REGION Network 79: CmFinalRollerFrontAxisX Position Absolute Position1
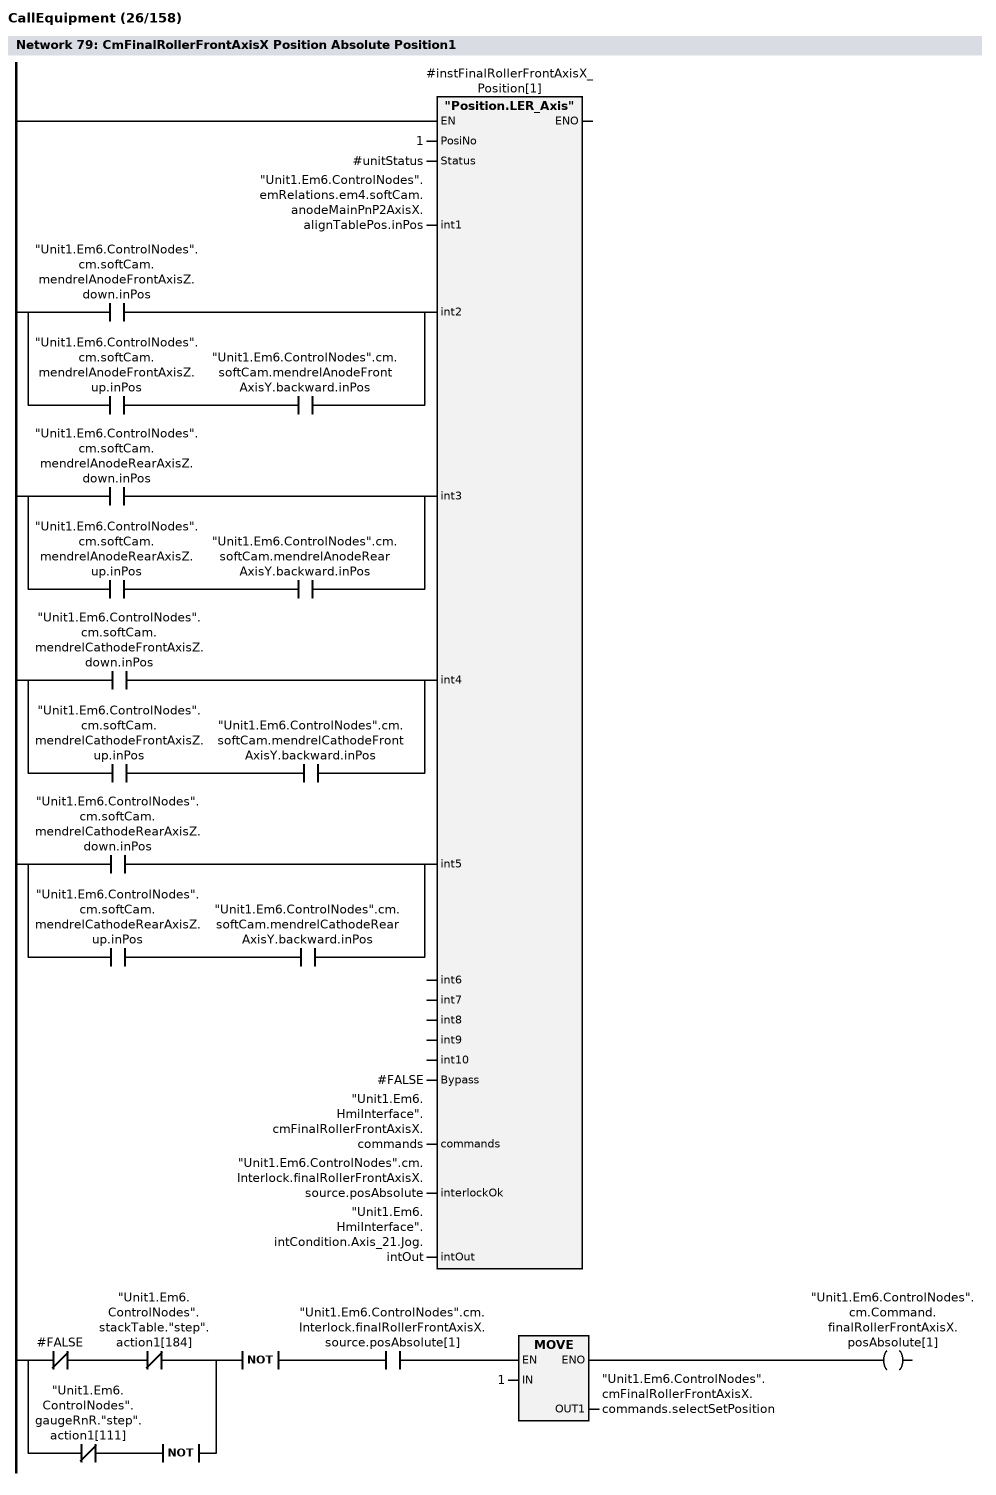
   RUNG wire#powerrail
      #instFinalRollerFrontAxisX_Position[1](int2 := wire#w1, int3 := wire#w2, int4 := wire#w3, int5 := wire#w4, PosiNo := 1, Status := #unitStatus, int1 := "Unit1.Em6.ControlNodes".emRelations.em4.softCam.anodeMainPnP2AxisX.alignTablePos.inPos, int6 :=, int7 :=, int8 :=, int9 :=, int10 :=, Bypass := #FALSE, commands := "Unit1.Em6.HmiInterface".cmFinalRollerFrontAxisX.commands, interlockOk := "Unit1.Em6.ControlNodes".cm.Interlock.finalRollerFrontAxisX.source.posAbsolute, intOut := "Unit1.Em6.HmiInterface".intCondition.Axis_21.Jog.intOut)
   END_RUNG
   RUNG wire#powerrail
      Contact( "Unit1.Em6.ControlNodes".cm.softCam.mendrelAnodeFrontAxisZ.down.inPos )
   END_RUNG wire#w1
   RUNG wire#powerrail
      Contact( "Unit1.Em6.ControlNodes".cm.softCam.mendrelAnodeFrontAxisZ.up.inPos )
      Contact( "Unit1.Em6.ControlNodes".cm.softCam.mendrelAnodeFrontAxisY.backward.inPos )
   END_RUNG wire#w1
   RUNG wire#powerrail
      Contact( "Unit1.Em6.ControlNodes".cm.softCam.mendrelAnodeRearAxisZ.down.inPos )
   END_RUNG wire#w2
   RUNG wire#powerrail
      Contact( "Unit1.Em6.ControlNodes".cm.softCam.mendrelAnodeRearAxisZ.up.inPos )
      Contact( "Unit1.Em6.ControlNodes".cm.softCam.mendrelAnodeRearAxisY.backward.inPos )
   END_RUNG wire#w2
   RUNG wire#powerrail
      Contact( "Unit1.Em6.ControlNodes".cm.softCam.mendrelCathodeFrontAxisZ.down.inPos )
   END_RUNG wire#w3
   RUNG wire#powerrail
      Contact( "Unit1.Em6.ControlNodes".cm.softCam.mendrelCathodeFrontAxisZ.up.inPos )
      Contact( "Unit1.Em6.ControlNodes".cm.softCam.mendrelCathodeFrontAxisY.backward.inPos )
   END_RUNG wire#w3
   RUNG wire#powerrail
      Contact( "Unit1.Em6.ControlNodes".cm.softCam.mendrelCathodeRearAxisZ.down.inPos )
   END_RUNG wire#w4
   RUNG wire#powerrail
      Contact( "Unit1.Em6.ControlNodes".cm.softCam.mendrelCathodeRearAxisZ.up.inPos )
      Contact( "Unit1.Em6.ControlNodes".cm.softCam.mendrelCathodeRearAxisY.backward.inPos )
   END_RUNG wire#w4
   RUNG wire#powerrail
      I_Contact( #FALSE )
      I_Contact( "Unit1.Em6.ControlNodes".stackTable."step".action1[184] )
      wire#w5
      Not()
      Contact( "Unit1.Em6.ControlNodes".cm.Interlock.finalRollerFrontAxisX.source.posAbsolute[1] )
      Move(in := 1, out1 => "Unit1.Em6.ControlNodes".cmFinalRollerFrontAxisX.commands.selectSetPosition)
      Coil( "Unit1.Em6.ControlNodes".cm.Command.finalRollerFrontAxisX.posAbsolute[1] )
   END_RUNG
   RUNG wire#powerrail
      I_Contact( "Unit1.Em6.ControlNodes".gaugeRnR."step".action1[111] )
      Not()
   END_RUNG wire#w5
   // the same network as SCL:
   #instFinalRollerFrontAxisX_Position[1](PosiNo := 1,   // "Position.LER_Axis"
                           Status := #unitStatus,
                           int1 := "Unit1.Em6.ControlNodes".emRelations.em4.softCam.anodeMainPnP2AxisX.alignTablePos.inPos,
                           int2 := "Unit1.Em6.ControlNodes".cm.softCam.mendrelAnodeFrontAxisZ.down.inPos OR ("Unit1.Em6.ControlNodes".cm.softCam.mendrelAnodeFrontAxisZ.up.inPos AND "Unit1.Em6.ControlNodes".cm.softCam.mendrelAnodeFrontAxisY.backward.inPos),
                           int3 := "Unit1.Em6.ControlNodes".cm.softCam.mendrelAnodeRearAxisZ.down.inPos OR ("Unit1.Em6.ControlNodes".cm.softCam.mendrelAnodeRearAxisZ.up.inPos AND "Unit1.Em6.ControlNodes".cm.softCam.mendrelAnodeRearAxisY.backward.inPos),
                           int4 := "Unit1.Em6.ControlNodes".cm.softCam.mendrelCathodeFrontAxisZ.down.inPos OR ("Unit1.Em6.ControlNodes".cm.softCam.mendrelCathodeFrontAxisZ.up.inPos AND "Unit1.Em6.ControlNodes".cm.softCam.mendrelCathodeFrontAxisY.backward.inPos),
                           int5 := "Unit1.Em6.ControlNodes".cm.softCam.mendrelCathodeRearAxisZ.down.inPos OR ("Unit1.Em6.ControlNodes".cm.softCam.mendrelCathodeRearAxisZ.up.inPos AND "Unit1.Em6.ControlNodes".cm.softCam.mendrelCathodeRearAxisY.backward.inPos),
                           Bypass := #FALSE,
                           commands := "Unit1.Em6.HmiInterface".cmFinalRollerFrontAxisX.commands,
                           interlockOk := "Unit1.Em6.ControlNodes".cm.Interlock.finalRollerFrontAxisX.source.posAbsolute,
                           intOut := "Unit1.Em6.HmiInterface".intCondition.Axis_21.Jog.intOut);
   #_w1 := NOT ((NOT #FALSE AND NOT "Unit1.Em6.ControlNodes".stackTable."step".action1[184]) OR NOT (NOT "Unit1.Em6.ControlNodes".gaugeRnR."step".action1[111])) AND "Unit1.Em6.ControlNodes".cm.Interlock.finalRollerFrontAxisX.source.posAbsolute[1];
   IF #_w1 THEN "Unit1.Em6.ControlNodes".cmFinalRollerFrontAxisX.commands.selectSetPosition := 1; END_IF;
   "Unit1.Em6.ControlNodes".cm.Command.finalRollerFrontAxisX.posAbsolute[1] := #_w1;
END_REGION

REGION Network 80: CmFinalRollerFrontAxisX Position Absolute Position2
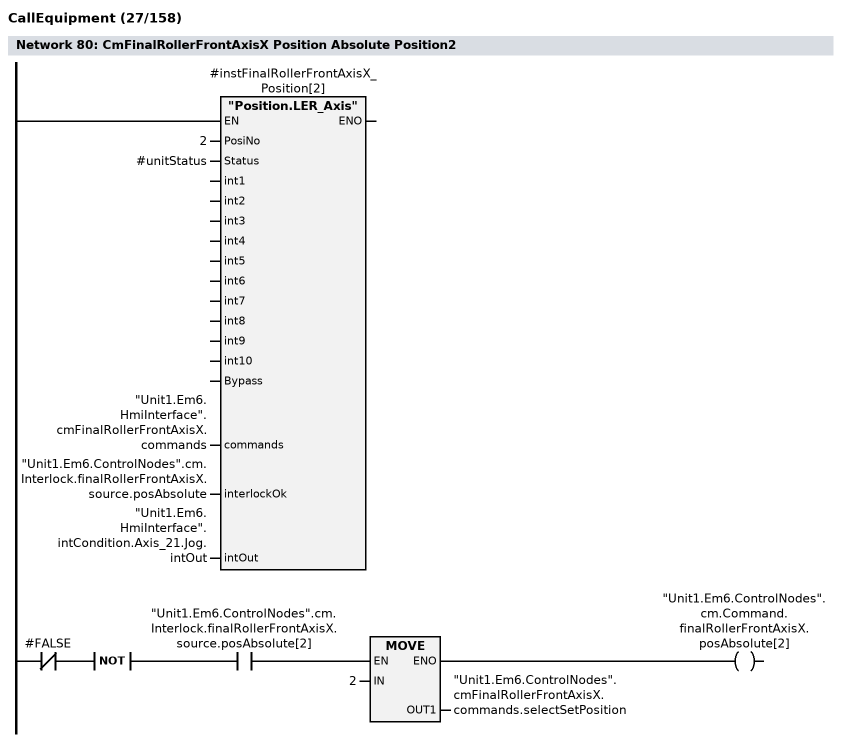
   RUNG wire#powerrail
      #instFinalRollerFrontAxisX_Position[2](PosiNo := 2, Status := #unitStatus, int1 :=, int2 :=, int3 :=, int4 :=, int5 :=, int6 :=, int7 :=, int8 :=, int9 :=, int10 :=, Bypass :=, commands := "Unit1.Em6.HmiInterface".cmFinalRollerFrontAxisX.commands, interlockOk := "Unit1.Em6.ControlNodes".cm.Interlock.finalRollerFrontAxisX.source.posAbsolute, intOut := "Unit1.Em6.HmiInterface".intCondition.Axis_21.Jog.intOut)
   END_RUNG
   RUNG wire#powerrail
      I_Contact( #FALSE )
      Not()
      Contact( "Unit1.Em6.ControlNodes".cm.Interlock.finalRollerFrontAxisX.source.posAbsolute[2] )
      Move(in := 2, out1 => "Unit1.Em6.ControlNodes".cmFinalRollerFrontAxisX.commands.selectSetPosition)
      Coil( "Unit1.Em6.ControlNodes".cm.Command.finalRollerFrontAxisX.posAbsolute[2] )
   END_RUNG
   // the same network as SCL:
   #instFinalRollerFrontAxisX_Position[2](PosiNo := 2,   // "Position.LER_Axis"
                           Status := #unitStatus,
                           commands := "Unit1.Em6.HmiInterface".cmFinalRollerFrontAxisX.commands,
                           interlockOk := "Unit1.Em6.ControlNodes".cm.Interlock.finalRollerFrontAxisX.source.posAbsolute,
                           intOut := "Unit1.Em6.HmiInterface".intCondition.Axis_21.Jog.intOut);
   #_w1 := NOT (NOT #FALSE) AND "Unit1.Em6.ControlNodes".cm.Interlock.finalRollerFrontAxisX.source.posAbsolute[2];
   IF #_w1 THEN "Unit1.Em6.ControlNodes".cmFinalRollerFrontAxisX.commands.selectSetPosition := 2; END_IF;
   "Unit1.Em6.ControlNodes".cm.Command.finalRollerFrontAxisX.posAbsolute[2] := #_w1;
END_REGION

REGION Network 81: CmFinalRollerFrontAxisX Position Absolute Position3
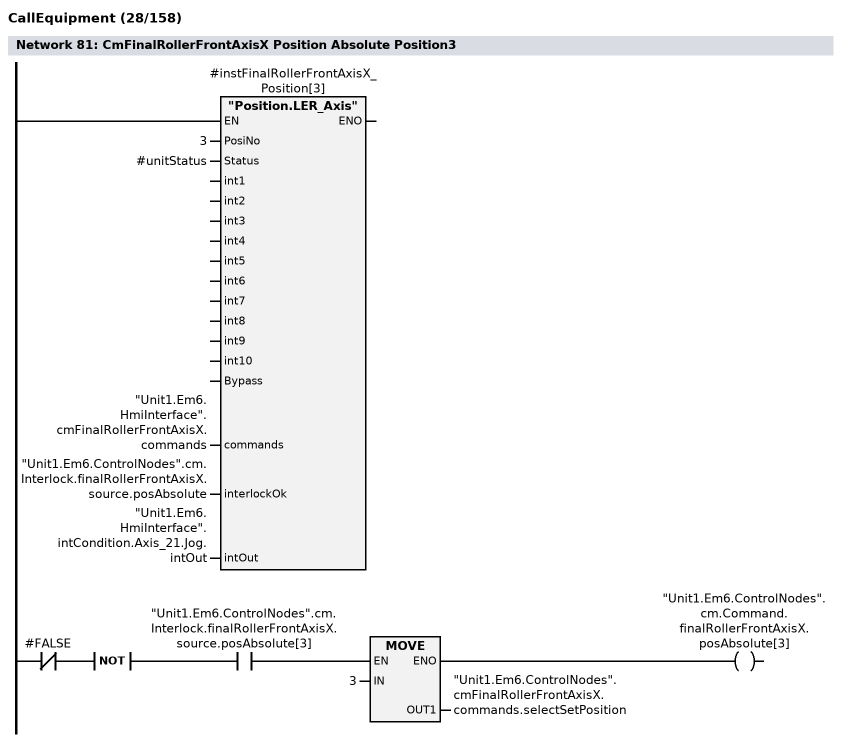
   RUNG wire#powerrail
      #instFinalRollerFrontAxisX_Position[3](PosiNo := 3, Status := #unitStatus, int1 :=, int2 :=, int3 :=, int4 :=, int5 :=, int6 :=, int7 :=, int8 :=, int9 :=, int10 :=, Bypass :=, commands := "Unit1.Em6.HmiInterface".cmFinalRollerFrontAxisX.commands, interlockOk := "Unit1.Em6.ControlNodes".cm.Interlock.finalRollerFrontAxisX.source.posAbsolute, intOut := "Unit1.Em6.HmiInterface".intCondition.Axis_21.Jog.intOut)
   END_RUNG
   RUNG wire#powerrail
      I_Contact( #FALSE )
      Not()
      Contact( "Unit1.Em6.ControlNodes".cm.Interlock.finalRollerFrontAxisX.source.posAbsolute[3] )
      Move(in := 3, out1 => "Unit1.Em6.ControlNodes".cmFinalRollerFrontAxisX.commands.selectSetPosition)
      Coil( "Unit1.Em6.ControlNodes".cm.Command.finalRollerFrontAxisX.posAbsolute[3] )
   END_RUNG
   // the same network as SCL:
   #instFinalRollerFrontAxisX_Position[3](PosiNo := 3,   // "Position.LER_Axis"
                           Status := #unitStatus,
                           commands := "Unit1.Em6.HmiInterface".cmFinalRollerFrontAxisX.commands,
                           interlockOk := "Unit1.Em6.ControlNodes".cm.Interlock.finalRollerFrontAxisX.source.posAbsolute,
                           intOut := "Unit1.Em6.HmiInterface".intCondition.Axis_21.Jog.intOut);
   #_w1 := NOT (NOT #FALSE) AND "Unit1.Em6.ControlNodes".cm.Interlock.finalRollerFrontAxisX.source.posAbsolute[3];
   IF #_w1 THEN "Unit1.Em6.ControlNodes".cmFinalRollerFrontAxisX.commands.selectSetPosition := 3; END_IF;
   "Unit1.Em6.ControlNodes".cm.Command.finalRollerFrontAxisX.posAbsolute[3] := #_w1;
END_REGION

REGION Network 82: CmFinalRollerFrontAxisX Position Absolute Position4
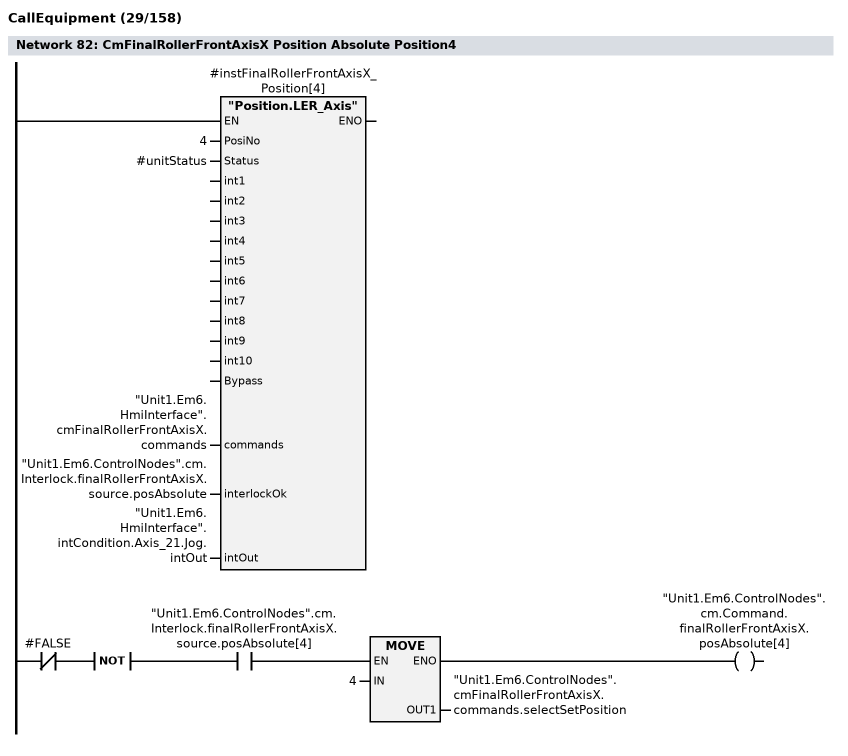
   RUNG wire#powerrail
      #instFinalRollerFrontAxisX_Position[4](PosiNo := 4, Status := #unitStatus, int1 :=, int2 :=, int3 :=, int4 :=, int5 :=, int6 :=, int7 :=, int8 :=, int9 :=, int10 :=, Bypass :=, commands := "Unit1.Em6.HmiInterface".cmFinalRollerFrontAxisX.commands, interlockOk := "Unit1.Em6.ControlNodes".cm.Interlock.finalRollerFrontAxisX.source.posAbsolute, intOut := "Unit1.Em6.HmiInterface".intCondition.Axis_21.Jog.intOut)
   END_RUNG
   RUNG wire#powerrail
      I_Contact( #FALSE )
      Not()
      Contact( "Unit1.Em6.ControlNodes".cm.Interlock.finalRollerFrontAxisX.source.posAbsolute[4] )
      Move(in := 4, out1 => "Unit1.Em6.ControlNodes".cmFinalRollerFrontAxisX.commands.selectSetPosition)
      Coil( "Unit1.Em6.ControlNodes".cm.Command.finalRollerFrontAxisX.posAbsolute[4] )
   END_RUNG
   // the same network as SCL:
   #instFinalRollerFrontAxisX_Position[4](PosiNo := 4,   // "Position.LER_Axis"
                           Status := #unitStatus,
                           commands := "Unit1.Em6.HmiInterface".cmFinalRollerFrontAxisX.commands,
                           interlockOk := "Unit1.Em6.ControlNodes".cm.Interlock.finalRollerFrontAxisX.source.posAbsolute,
                           intOut := "Unit1.Em6.HmiInterface".intCondition.Axis_21.Jog.intOut);
   #_w1 := NOT (NOT #FALSE) AND "Unit1.Em6.ControlNodes".cm.Interlock.finalRollerFrontAxisX.source.posAbsolute[4];
   IF #_w1 THEN "Unit1.Em6.ControlNodes".cmFinalRollerFrontAxisX.commands.selectSetPosition := 4; END_IF;
   "Unit1.Em6.ControlNodes".cm.Command.finalRollerFrontAxisX.posAbsolute[4] := #_w1;
END_REGION

REGION Network 83: CmFinalRollerFrontAxisX Position Absolute Position5
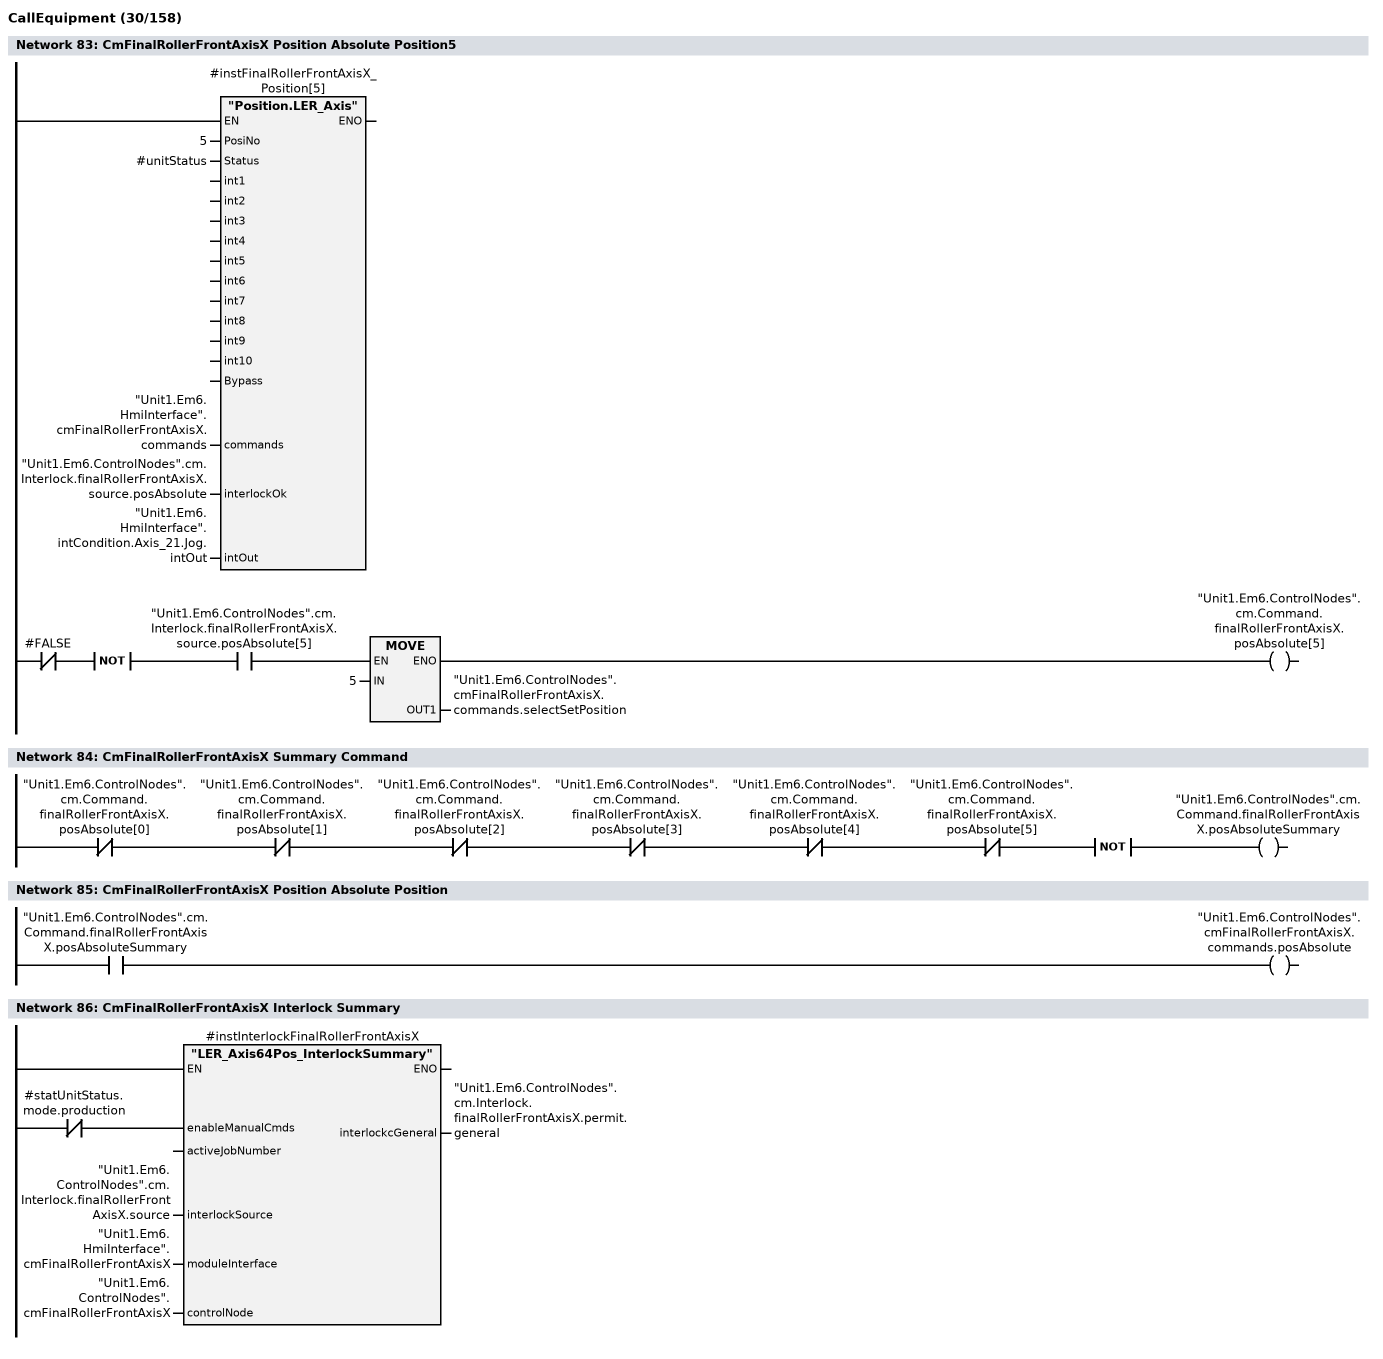
   RUNG wire#powerrail
      #instFinalRollerFrontAxisX_Position[5](PosiNo := 5, Status := #unitStatus, int1 :=, int2 :=, int3 :=, int4 :=, int5 :=, int6 :=, int7 :=, int8 :=, int9 :=, int10 :=, Bypass :=, commands := "Unit1.Em6.HmiInterface".cmFinalRollerFrontAxisX.commands, interlockOk := "Unit1.Em6.ControlNodes".cm.Interlock.finalRollerFrontAxisX.source.posAbsolute, intOut := "Unit1.Em6.HmiInterface".intCondition.Axis_21.Jog.intOut)
   END_RUNG
   RUNG wire#powerrail
      I_Contact( #FALSE )
      Not()
      Contact( "Unit1.Em6.ControlNodes".cm.Interlock.finalRollerFrontAxisX.source.posAbsolute[5] )
      Move(in := 5, out1 => "Unit1.Em6.ControlNodes".cmFinalRollerFrontAxisX.commands.selectSetPosition)
      Coil( "Unit1.Em6.ControlNodes".cm.Command.finalRollerFrontAxisX.posAbsolute[5] )
   END_RUNG
   // the same network as SCL:
   #instFinalRollerFrontAxisX_Position[5](PosiNo := 5,   // "Position.LER_Axis"
                           Status := #unitStatus,
                           commands := "Unit1.Em6.HmiInterface".cmFinalRollerFrontAxisX.commands,
                           interlockOk := "Unit1.Em6.ControlNodes".cm.Interlock.finalRollerFrontAxisX.source.posAbsolute,
                           intOut := "Unit1.Em6.HmiInterface".intCondition.Axis_21.Jog.intOut);
   #_w1 := NOT (NOT #FALSE) AND "Unit1.Em6.ControlNodes".cm.Interlock.finalRollerFrontAxisX.source.posAbsolute[5];
   IF #_w1 THEN "Unit1.Em6.ControlNodes".cmFinalRollerFrontAxisX.commands.selectSetPosition := 5; END_IF;
   "Unit1.Em6.ControlNodes".cm.Command.finalRollerFrontAxisX.posAbsolute[5] := #_w1;
END_REGION

REGION Network 84: CmFinalRollerFrontAxisX Summary Command
   RUNG wire#powerrail
      I_Contact( "Unit1.Em6.ControlNodes".cm.Command.finalRollerFrontAxisX.posAbsolute[0] )
      I_Contact( "Unit1.Em6.ControlNodes".cm.Command.finalRollerFrontAxisX.posAbsolute[1] )
      I_Contact( "Unit1.Em6.ControlNodes".cm.Command.finalRollerFrontAxisX.posAbsolute[2] )
      I_Contact( "Unit1.Em6.ControlNodes".cm.Command.finalRollerFrontAxisX.posAbsolute[3] )
      I_Contact( "Unit1.Em6.ControlNodes".cm.Command.finalRollerFrontAxisX.posAbsolute[4] )
      I_Contact( "Unit1.Em6.ControlNodes".cm.Command.finalRollerFrontAxisX.posAbsolute[5] )
      Not()
      Coil( "Unit1.Em6.ControlNodes".cm.Command.finalRollerFrontAxisX.posAbsoluteSummary )
   END_RUNG
   // the same network as SCL:
   "Unit1.Em6.ControlNodes".cm.Command.finalRollerFrontAxisX.posAbsoluteSummary := NOT (NOT "Unit1.Em6.ControlNodes".cm.Command.finalRollerFrontAxisX.posAbsolute[0] AND NOT "Unit1.Em6.ControlNodes".cm.Command.finalRollerFrontAxisX.posAbsolute[1] AND NOT "Unit1.Em6.ControlNodes".cm.Command.finalRollerFrontAxisX.posAbsolute[2] AND NOT "Unit1.Em6.ControlNodes".cm.Command.finalRollerFrontAxisX.posAbsolute[3] AND NOT "Unit1.Em6.ControlNodes".cm.Command.finalRollerFrontAxisX.posAbsolute[4] AND NOT "Unit1.Em6.ControlNodes".cm.Command.finalRollerFrontAxisX.posAbsolute[5]);
END_REGION

REGION Network 85: CmFinalRollerFrontAxisX Position Absolute Position
   RUNG wire#powerrail
      Contact( "Unit1.Em6.ControlNodes".cm.Command.finalRollerFrontAxisX.posAbsoluteSummary )
      Coil( "Unit1.Em6.ControlNodes".cmFinalRollerFrontAxisX.commands.posAbsolute )
   END_RUNG
   // the same network as SCL:
   "Unit1.Em6.ControlNodes".cmFinalRollerFrontAxisX.commands.posAbsolute := "Unit1.Em6.ControlNodes".cm.Command.finalRollerFrontAxisX.posAbsoluteSummary;
END_REGION

REGION Network 86: CmFinalRollerFrontAxisX Interlock Summary
   RUNG wire#powerrail
      #instInterlockFinalRollerFrontAxisX(enableManualCmds := wire#w1, activeJobNumber :=, interlockSource := "Unit1.Em6.ControlNodes".cm.Interlock.finalRollerFrontAxisX.source, moduleInterface := "Unit1.Em6.HmiInterface".cmFinalRollerFrontAxisX, controlNode := "Unit1.Em6.ControlNodes".cmFinalRollerFrontAxisX, interlockcGeneral => "Unit1.Em6.ControlNodes".cm.Interlock.finalRollerFrontAxisX.permit.general)
   END_RUNG
   RUNG wire#powerrail
      I_Contact( #statUnitStatus.mode.production )
   END_RUNG wire#w1
   // the same network as SCL:
   #instInterlockFinalRollerFrontAxisX(enableManualCmds := NOT #statUnitStatus.mode.production,   // "LER_Axis64Pos_InterlockSummary"
                           interlockSource := "Unit1.Em6.ControlNodes".cm.Interlock.finalRollerFrontAxisX.source,
                           moduleInterface := "Unit1.Em6.HmiInterface".cmFinalRollerFrontAxisX,
                           controlNode := "Unit1.Em6.ControlNodes".cmFinalRollerFrontAxisX,
                           interlockcGeneral => "Unit1.Em6.ControlNodes".cm.Interlock.finalRollerFrontAxisX.permit.general);
END_REGION

REGION Network 87: CmFinalRollerFrontAxisX velocity/speed
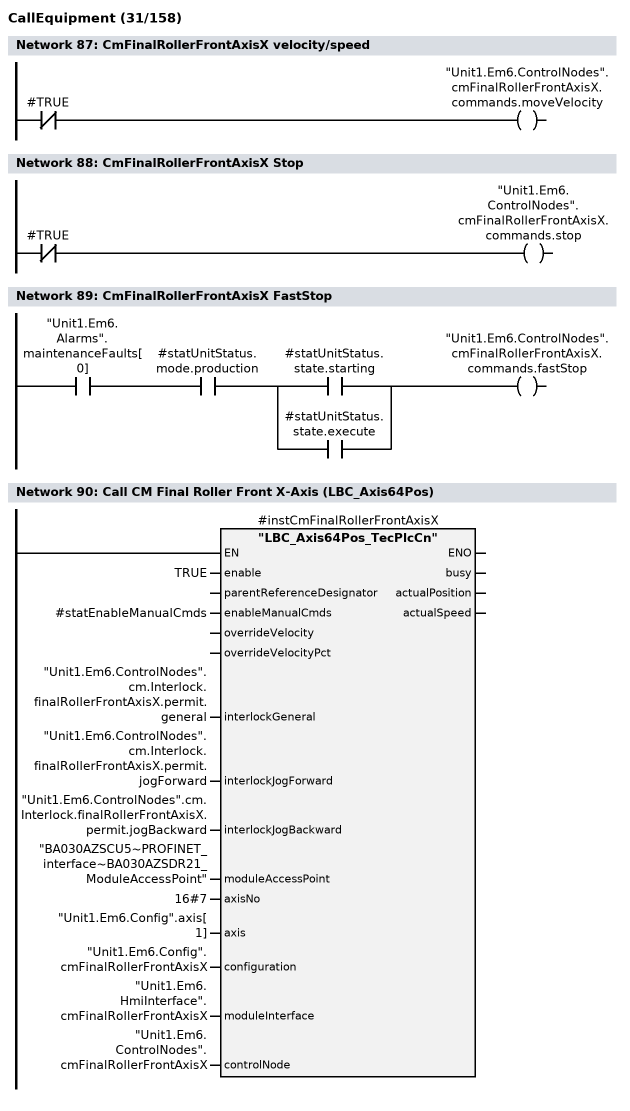
   RUNG wire#powerrail
      I_Contact( #TRUE )
      Coil( "Unit1.Em6.ControlNodes".cmFinalRollerFrontAxisX.commands.moveVelocity )
   END_RUNG
   // the same network as SCL:
   "Unit1.Em6.ControlNodes".cmFinalRollerFrontAxisX.commands.moveVelocity := NOT #TRUE;
END_REGION

REGION Network 88: CmFinalRollerFrontAxisX Stop
   RUNG wire#powerrail
      I_Contact( #TRUE )
      Coil( "Unit1.Em6.ControlNodes".cmFinalRollerFrontAxisX.commands.stop )
   END_RUNG
   // the same network as SCL:
   "Unit1.Em6.ControlNodes".cmFinalRollerFrontAxisX.commands.stop := NOT #TRUE;
END_REGION

REGION Network 89: CmFinalRollerFrontAxisX FastStop
   RUNG wire#powerrail
      Contact( "Unit1.Em6.Alarms".maintenanceFaults[0] )
      Contact( #statUnitStatus.mode.production )
      wire#w1
      Contact( #statUnitStatus.state.starting )
      wire#w2
      Coil( "Unit1.Em6.ControlNodes".cmFinalRollerFrontAxisX.commands.fastStop )
   END_RUNG
   RUNG wire#w1
      Contact( #statUnitStatus.state.execute )
   END_RUNG wire#w2
   // the same network as SCL:
   "Unit1.Em6.ControlNodes".cmFinalRollerFrontAxisX.commands.fastStop := "Unit1.Em6.Alarms".maintenanceFaults[0] AND #statUnitStatus.mode.production AND (#statUnitStatus.state.starting OR #statUnitStatus.state.execute);
END_REGION

REGION Network 90: Call CM Final Roller Front X-Axis (LBC_Axis64Pos)
   RUNG wire#powerrail
      #instCmFinalRollerFrontAxisX(enable := TRUE, parentReferenceDesignator :=, enableManualCmds := #statEnableManualCmds, overrideVelocity :=, overrideVelocityPct :=, interlockGeneral := "Unit1.Em6.ControlNodes".cm.Interlock.finalRollerFrontAxisX.permit.general, interlockJogForward := "Unit1.Em6.ControlNodes".cm.Interlock.finalRollerFrontAxisX.permit.jogForward, interlockJogBackward := "Unit1.Em6.ControlNodes".cm.Interlock.finalRollerFrontAxisX.permit.jogBackward, moduleAccessPoint := "BA030AZSCU5~PROFINET_interface~BA030AZSDR21_ModuleAccessPoint", axisNo := 16#7, axis := "Unit1.Em6.Config".axis[1], configuration := "Unit1.Em6.Config".cmFinalRollerFrontAxisX, moduleInterface := "Unit1.Em6.HmiInterface".cmFinalRollerFrontAxisX, controlNode := "Unit1.Em6.ControlNodes".cmFinalRollerFrontAxisX, busy =>, actualPosition =>, actualSpeed =>)
   END_RUNG
   // the same network as SCL:
   #instCmFinalRollerFrontAxisX(enable := TRUE,   // "LBC_Axis64Pos_TecPlcCn"
                           enableManualCmds := #statEnableManualCmds,
                           interlockGeneral := "Unit1.Em6.ControlNodes".cm.Interlock.finalRollerFrontAxisX.permit.general,
                           interlockJogForward := "Unit1.Em6.ControlNodes".cm.Interlock.finalRollerFrontAxisX.permit.jogForward,
                           interlockJogBackward := "Unit1.Em6.ControlNodes".cm.Interlock.finalRollerFrontAxisX.permit.jogBackward,
                           moduleAccessPoint := "BA030AZSCU5~PROFINET_interface~BA030AZSDR21_ModuleAccessPoint",
                           axisNo := 16#7,
                           axis := "Unit1.Em6.Config".axis[1],
                           configuration := "Unit1.Em6.Config".cmFinalRollerFrontAxisX,
                           moduleInterface := "Unit1.Em6.HmiInterface".cmFinalRollerFrontAxisX,
                           controlNode := "Unit1.Em6.ControlNodes".cmFinalRollerFrontAxisX);
END_REGION

REGION Network 91: CmCathodeMainPnP1AxisX SoftCam
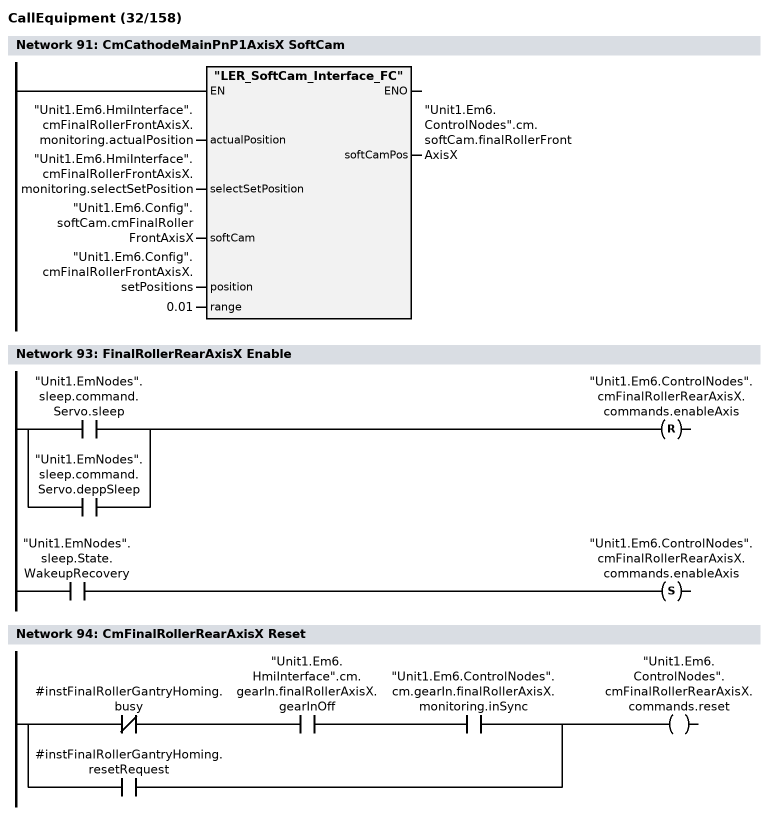
   RUNG wire#powerrail
      "LER_SoftCam_Interface_FC"(actualPosition := "Unit1.Em6.HmiInterface".cmFinalRollerFrontAxisX.monitoring.actualPosition, selectSetPosition := "Unit1.Em6.HmiInterface".cmFinalRollerFrontAxisX.monitoring.selectSetPosition, softCam := "Unit1.Em6.Config".softCam.cmFinalRollerFrontAxisX, position := "Unit1.Em6.Config".cmFinalRollerFrontAxisX.setPositions, range := 0.01, softCamPos => "Unit1.Em6.ControlNodes".cm.softCam.finalRollerFrontAxisX)
   END_RUNG
   // the same network as SCL:
   "LER_SoftCam_Interface_FC"(actualPosition := "Unit1.Em6.HmiInterface".cmFinalRollerFrontAxisX.monitoring.actualPosition,
                           selectSetPosition := "Unit1.Em6.HmiInterface".cmFinalRollerFrontAxisX.monitoring.selectSetPosition,
                           softCam := "Unit1.Em6.Config".softCam.cmFinalRollerFrontAxisX,
                           position := "Unit1.Em6.Config".cmFinalRollerFrontAxisX.setPositions,
                           range := 0.01,
                           softCamPos => "Unit1.Em6.ControlNodes".cm.softCam.finalRollerFrontAxisX);
END_REGION

REGION Network 93: FinalRollerRearAxisX Enable
   RUNG wire#powerrail
      Contact( "Unit1.EmNodes".sleep.command.Servo.sleep )
      wire#w1
      R_Coil( "Unit1.Em6.ControlNodes".cmFinalRollerRearAxisX.commands.enableAxis )
   END_RUNG
   RUNG wire#powerrail
      Contact( "Unit1.EmNodes".sleep.command.Servo.deppSleep )
   END_RUNG wire#w1
   RUNG wire#powerrail
      Contact( "Unit1.EmNodes".sleep.State.WakeupRecovery )
      S_Coil( "Unit1.Em6.ControlNodes".cmFinalRollerRearAxisX.commands.enableAxis )
   END_RUNG
   // the same network as SCL:
   IF "Unit1.EmNodes".sleep.command.Servo.sleep OR "Unit1.EmNodes".sleep.command.Servo.deppSleep THEN
       "Unit1.Em6.ControlNodes".cmFinalRollerRearAxisX.commands.enableAxis := FALSE;
   END_IF;
   IF "Unit1.EmNodes".sleep.State.WakeupRecovery THEN
       "Unit1.Em6.ControlNodes".cmFinalRollerRearAxisX.commands.enableAxis := TRUE;
   END_IF;
END_REGION

REGION Network 94: CmFinalRollerRearAxisX Reset
   RUNG wire#powerrail
      I_Contact( #instFinalRollerGantryHoming.busy )
      Contact( "Unit1.Em6.HmiInterface".cm.gearIn.finalRollerAxisX.gearInOff )
      Contact( "Unit1.Em6.ControlNodes".cm.gearIn.finalRollerAxisX.monitoring.inSync )
      wire#w1
      Coil( "Unit1.Em6.ControlNodes".cmFinalRollerRearAxisX.commands.reset )
   END_RUNG
   RUNG wire#powerrail
      Contact( #instFinalRollerGantryHoming.resetRequest )
   END_RUNG wire#w1
   // the same network as SCL:
   "Unit1.Em6.ControlNodes".cmFinalRollerRearAxisX.commands.reset := (NOT #instFinalRollerGantryHoming.busy AND "Unit1.Em6.HmiInterface".cm.gearIn.finalRollerAxisX.gearInOff AND "Unit1.Em6.ControlNodes".cm.gearIn.finalRollerAxisX.monitoring.inSync) OR #instFinalRollerGantryHoming.resetRequest;
END_REGION

REGION Network 95: CmFinalRollerRearAxisX Home
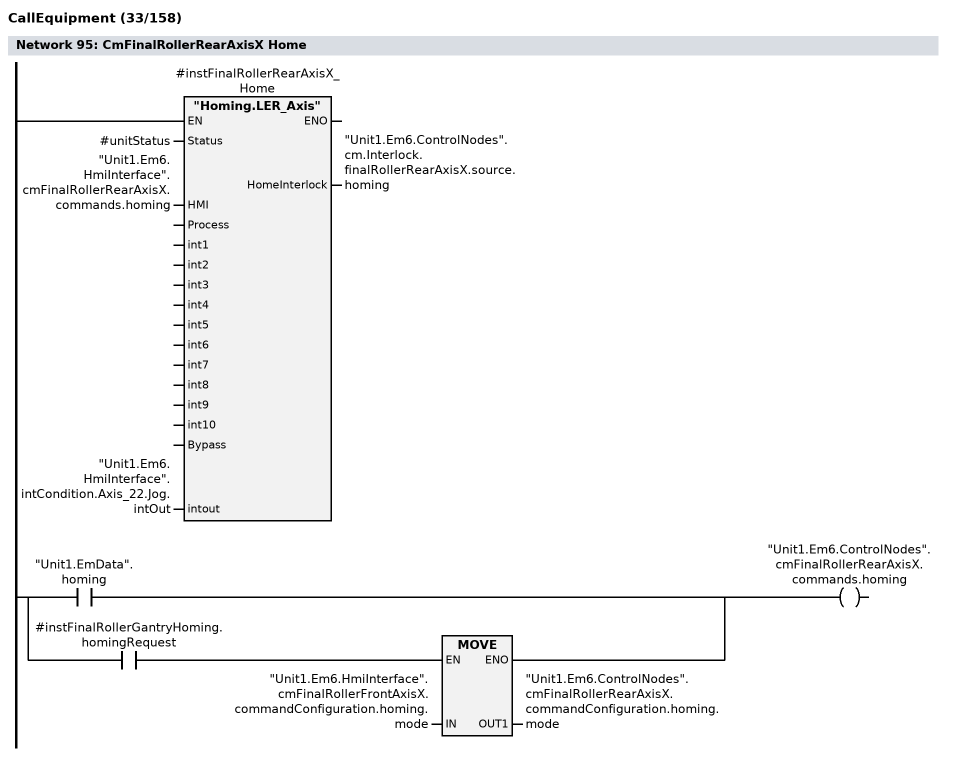
   RUNG wire#powerrail
      #instFinalRollerRearAxisX_Home(Status := #unitStatus, HMI := "Unit1.Em6.HmiInterface".cmFinalRollerRearAxisX.commands.homing, Process :=, int1 :=, int2 :=, int3 :=, int4 :=, int5 :=, int6 :=, int7 :=, int8 :=, int9 :=, int10 :=, Bypass :=, intout := "Unit1.Em6.HmiInterface".intCondition.Axis_22.Jog.intOut, HomeInterlock => "Unit1.Em6.ControlNodes".cm.Interlock.finalRollerRearAxisX.source.homing)
   END_RUNG
   RUNG wire#powerrail
      Contact( "Unit1.EmData".homing )
      wire#w1
      Coil( "Unit1.Em6.ControlNodes".cmFinalRollerRearAxisX.commands.homing )
   END_RUNG
   RUNG wire#powerrail
      Contact( #instFinalRollerGantryHoming.homingRequest )
      Move(in := "Unit1.Em6.HmiInterface".cmFinalRollerFrontAxisX.commandConfiguration.homing.mode, out1 => "Unit1.Em6.ControlNodes".cmFinalRollerRearAxisX.commandConfiguration.homing.mode)
   END_RUNG wire#w1
   // the same network as SCL:
   #instFinalRollerRearAxisX_Home(Status := #unitStatus,   // "Homing.LER_Axis"
                           HMI := "Unit1.Em6.HmiInterface".cmFinalRollerRearAxisX.commands.homing,
                           intout := "Unit1.Em6.HmiInterface".intCondition.Axis_22.Jog.intOut,
                           HomeInterlock => "Unit1.Em6.ControlNodes".cm.Interlock.finalRollerRearAxisX.source.homing);
   IF #instFinalRollerGantryHoming.homingRequest THEN
       "Unit1.Em6.ControlNodes".cmFinalRollerRearAxisX.commandConfiguration.homing.mode := "Unit1.Em6.HmiInterface".cmFinalRollerFrontAxisX.commandConfiguration.homing.mode;
   END_IF;
   "Unit1.Em6.ControlNodes".cmFinalRollerRearAxisX.commands.homing := "Unit1.EmData".homing OR #instFinalRollerGantryHoming.homingRequest;
END_REGION

REGION Network 96: CmFinalRollerRearAxisX Position Absolute Jog
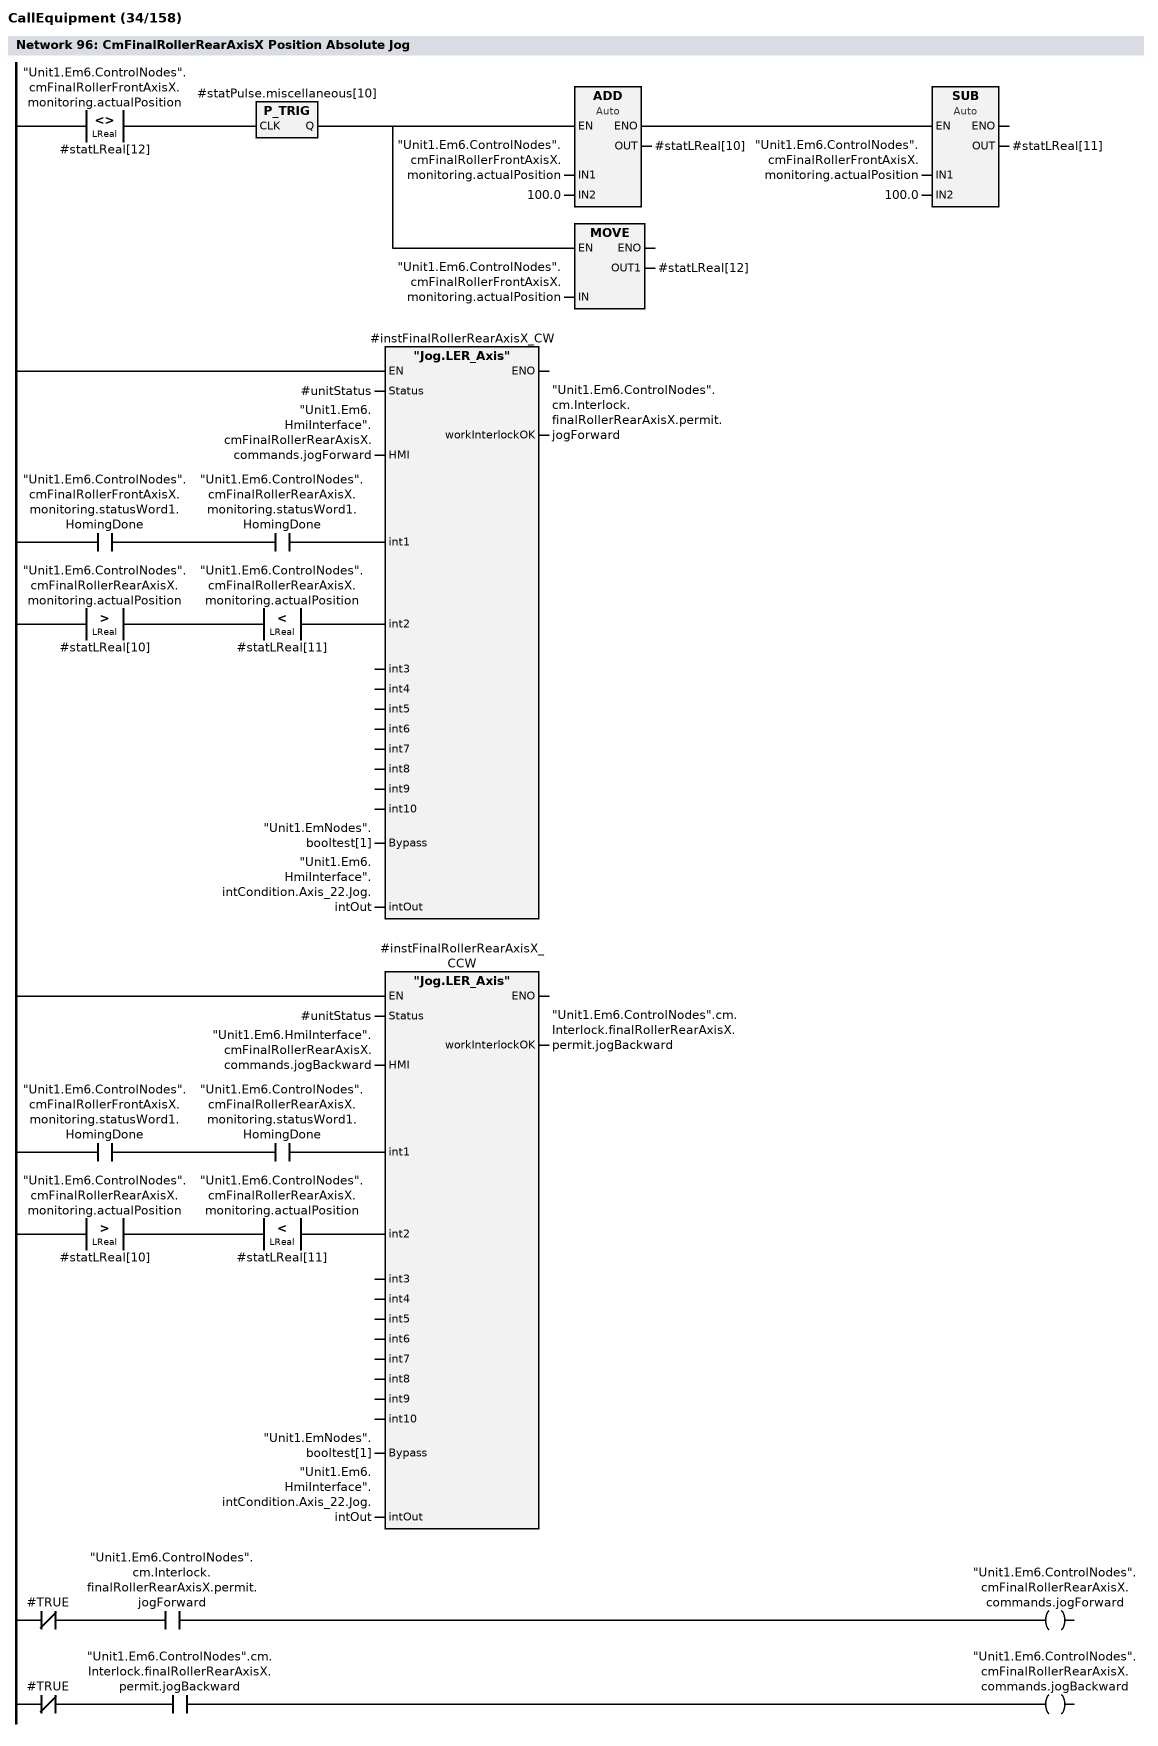
   RUNG wire#powerrail
      { S7_Templates := "SrcType := LReal" } NE_Contact(in1 := "Unit1.Em6.ControlNodes".cmFinalRollerFrontAxisX.monitoring.actualPosition, in2 := #statLReal[12])
      P_Trig( #statPulse.miscellaneous[10] )
      wire#w1
      Add(in1 := "Unit1.Em6.ControlNodes".cmFinalRollerFrontAxisX.monitoring.actualPosition, in2 := 100.0, out => #statLReal[10])
      Sub(in1 := "Unit1.Em6.ControlNodes".cmFinalRollerFrontAxisX.monitoring.actualPosition, in2 := 100.0, out => #statLReal[11])
   END_RUNG
   RUNG wire#w1
      Move(in := "Unit1.Em6.ControlNodes".cmFinalRollerFrontAxisX.monitoring.actualPosition, out1 => #statLReal[12])
   END_RUNG
   RUNG wire#powerrail
      #instFinalRollerRearAxisX_CW(int1 := wire#w2, int2 := wire#w3, Status := #unitStatus, HMI := "Unit1.Em6.HmiInterface".cmFinalRollerRearAxisX.commands.jogForward, int3 :=, int4 :=, int5 :=, int6 :=, int7 :=, int8 :=, int9 :=, int10 :=, Bypass := "Unit1.EmNodes".booltest[1], intOut := "Unit1.Em6.HmiInterface".intCondition.Axis_22.Jog.intOut, workInterlockOK => "Unit1.Em6.ControlNodes".cm.Interlock.finalRollerRearAxisX.permit.jogForward)
   END_RUNG
   RUNG wire#powerrail
      Contact( "Unit1.Em6.ControlNodes".cmFinalRollerFrontAxisX.monitoring.statusWord1.HomingDone )
      Contact( "Unit1.Em6.ControlNodes".cmFinalRollerRearAxisX.monitoring.statusWord1.HomingDone )
   END_RUNG wire#w2
   RUNG wire#powerrail
      { S7_Templates := "SrcType := LReal" } GT_Contact(in1 := "Unit1.Em6.ControlNodes".cmFinalRollerRearAxisX.monitoring.actualPosition, in2 := #statLReal[10])
      { S7_Templates := "SrcType := LReal" } LT_Contact(in1 := "Unit1.Em6.ControlNodes".cmFinalRollerRearAxisX.monitoring.actualPosition, in2 := #statLReal[11])
   END_RUNG wire#w3
   RUNG wire#powerrail
      #instFinalRollerRearAxisX_CCW(int1 := wire#w4, int2 := wire#w5, Status := #unitStatus, HMI := "Unit1.Em6.HmiInterface".cmFinalRollerRearAxisX.commands.jogBackward, int3 :=, int4 :=, int5 :=, int6 :=, int7 :=, int8 :=, int9 :=, int10 :=, Bypass := "Unit1.EmNodes".booltest[1], intOut := "Unit1.Em6.HmiInterface".intCondition.Axis_22.Jog.intOut, workInterlockOK => "Unit1.Em6.ControlNodes".cm.Interlock.finalRollerRearAxisX.permit.jogBackward)
   END_RUNG
   RUNG wire#powerrail
      Contact( "Unit1.Em6.ControlNodes".cmFinalRollerFrontAxisX.monitoring.statusWord1.HomingDone )
      Contact( "Unit1.Em6.ControlNodes".cmFinalRollerRearAxisX.monitoring.statusWord1.HomingDone )
   END_RUNG wire#w4
   RUNG wire#powerrail
      { S7_Templates := "SrcType := LReal" } GT_Contact(in1 := "Unit1.Em6.ControlNodes".cmFinalRollerRearAxisX.monitoring.actualPosition, in2 := #statLReal[10])
      { S7_Templates := "SrcType := LReal" } LT_Contact(in1 := "Unit1.Em6.ControlNodes".cmFinalRollerRearAxisX.monitoring.actualPosition, in2 := #statLReal[11])
   END_RUNG wire#w5
   RUNG wire#powerrail
      I_Contact( #TRUE )
      Contact( "Unit1.Em6.ControlNodes".cm.Interlock.finalRollerRearAxisX.permit.jogForward )
      Coil( "Unit1.Em6.ControlNodes".cmFinalRollerRearAxisX.commands.jogForward )
   END_RUNG
   RUNG wire#powerrail
      I_Contact( #TRUE )
      Contact( "Unit1.Em6.ControlNodes".cm.Interlock.finalRollerRearAxisX.permit.jogBackward )
      Coil( "Unit1.Em6.ControlNodes".cmFinalRollerRearAxisX.commands.jogBackward )
   END_RUNG
   // the same network as SCL:
   #_w1 := "Unit1.Em6.ControlNodes".cmFinalRollerFrontAxisX.monitoring.actualPosition <> #statLReal[12];
   #_w2 := #_w1 AND NOT #statPulse.miscellaneous[10];   // rising edge
   #statPulse.miscellaneous[10] := #_w1;
   IF #_w2 THEN
       #statLReal[10] := "Unit1.Em6.ControlNodes".cmFinalRollerFrontAxisX.monitoring.actualPosition + 100.0;
       #statLReal[11] := "Unit1.Em6.ControlNodes".cmFinalRollerFrontAxisX.monitoring.actualPosition - 100.0;
       #statLReal[12] := "Unit1.Em6.ControlNodes".cmFinalRollerFrontAxisX.monitoring.actualPosition;
   END_IF;
   #instFinalRollerRearAxisX_CW(Status := #unitStatus,   // "Jog.LER_Axis"
                           HMI := "Unit1.Em6.HmiInterface".cmFinalRollerRearAxisX.commands.jogForward,
                           int1 := "Unit1.Em6.ControlNodes".cmFinalRollerFrontAxisX.monitoring.statusWord1.HomingDone AND "Unit1.Em6.ControlNodes".cmFinalRollerRearAxisX.monitoring.statusWord1.HomingDone,
                           int2 := ("Unit1.Em6.ControlNodes".cmFinalRollerRearAxisX.monitoring.actualPosition > #statLReal[10]) AND ("Unit1.Em6.ControlNodes".cmFinalRollerRearAxisX.monitoring.actualPosition < #statLReal[11]),
                           Bypass := "Unit1.EmNodes".booltest[1],
                           intOut := "Unit1.Em6.HmiInterface".intCondition.Axis_22.Jog.intOut,
                           workInterlockOK => "Unit1.Em6.ControlNodes".cm.Interlock.finalRollerRearAxisX.permit.jogForward);
   #instFinalRollerRearAxisX_CCW(Status := #unitStatus,   // "Jog.LER_Axis"
                           HMI := "Unit1.Em6.HmiInterface".cmFinalRollerRearAxisX.commands.jogBackward,
                           int1 := "Unit1.Em6.ControlNodes".cmFinalRollerFrontAxisX.monitoring.statusWord1.HomingDone AND "Unit1.Em6.ControlNodes".cmFinalRollerRearAxisX.monitoring.statusWord1.HomingDone,
                           int2 := ("Unit1.Em6.ControlNodes".cmFinalRollerRearAxisX.monitoring.actualPosition > #statLReal[10]) AND ("Unit1.Em6.ControlNodes".cmFinalRollerRearAxisX.monitoring.actualPosition < #statLReal[11]),
                           Bypass := "Unit1.EmNodes".booltest[1],
                           intOut := "Unit1.Em6.HmiInterface".intCondition.Axis_22.Jog.intOut,
                           workInterlockOK => "Unit1.Em6.ControlNodes".cm.Interlock.finalRollerRearAxisX.permit.jogBackward);
   "Unit1.Em6.ControlNodes".cmFinalRollerRearAxisX.commands.jogForward := NOT #TRUE AND "Unit1.Em6.ControlNodes".cm.Interlock.finalRollerRearAxisX.permit.jogForward;
   "Unit1.Em6.ControlNodes".cmFinalRollerRearAxisX.commands.jogBackward := NOT #TRUE AND "Unit1.Em6.ControlNodes".cm.Interlock.finalRollerRearAxisX.permit.jogBackward;
END_REGION

REGION Network 97: CmFinalRollerRearAxisX Position Absolute Position0
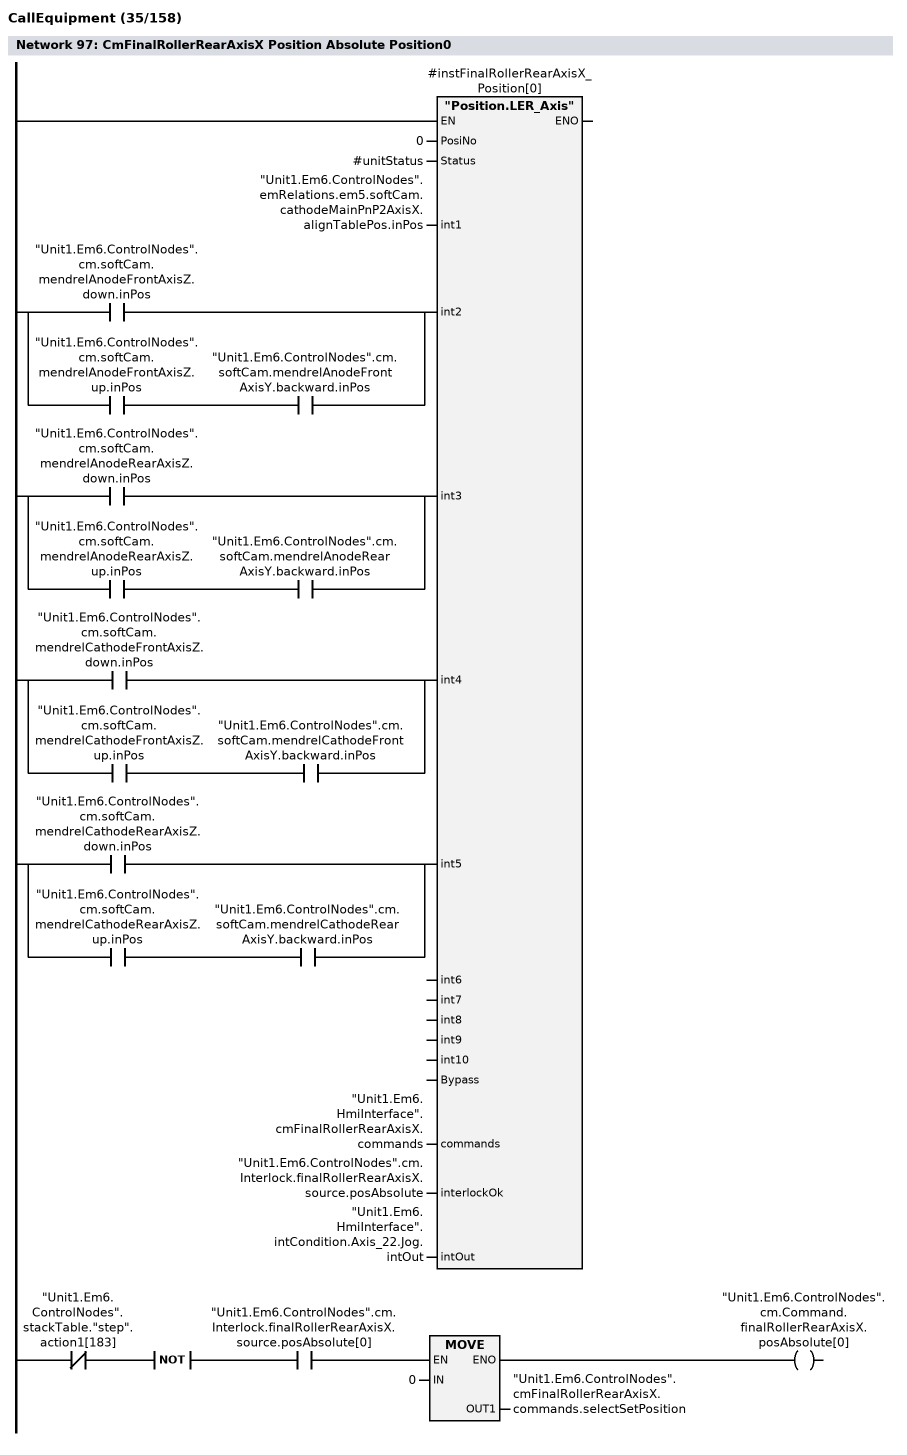
   RUNG wire#powerrail
      #instFinalRollerRearAxisX_Position[0](int2 := wire#w1, int3 := wire#w2, int4 := wire#w3, int5 := wire#w4, PosiNo := 0, Status := #unitStatus, int1 := "Unit1.Em6.ControlNodes".emRelations.em5.softCam.cathodeMainPnP2AxisX.alignTablePos.inPos, int6 :=, int7 :=, int8 :=, int9 :=, int10 :=, Bypass :=, commands := "Unit1.Em6.HmiInterface".cmFinalRollerRearAxisX.commands, interlockOk := "Unit1.Em6.ControlNodes".cm.Interlock.finalRollerRearAxisX.source.posAbsolute, intOut := "Unit1.Em6.HmiInterface".intCondition.Axis_22.Jog.intOut)
   END_RUNG
   RUNG wire#powerrail
      Contact( "Unit1.Em6.ControlNodes".cm.softCam.mendrelAnodeFrontAxisZ.down.inPos )
   END_RUNG wire#w1
   RUNG wire#powerrail
      Contact( "Unit1.Em6.ControlNodes".cm.softCam.mendrelAnodeFrontAxisZ.up.inPos )
      Contact( "Unit1.Em6.ControlNodes".cm.softCam.mendrelAnodeFrontAxisY.backward.inPos )
   END_RUNG wire#w1
   RUNG wire#powerrail
      Contact( "Unit1.Em6.ControlNodes".cm.softCam.mendrelAnodeRearAxisZ.down.inPos )
   END_RUNG wire#w2
   RUNG wire#powerrail
      Contact( "Unit1.Em6.ControlNodes".cm.softCam.mendrelAnodeRearAxisZ.up.inPos )
      Contact( "Unit1.Em6.ControlNodes".cm.softCam.mendrelAnodeRearAxisY.backward.inPos )
   END_RUNG wire#w2
   RUNG wire#powerrail
      Contact( "Unit1.Em6.ControlNodes".cm.softCam.mendrelCathodeFrontAxisZ.down.inPos )
   END_RUNG wire#w3
   RUNG wire#powerrail
      Contact( "Unit1.Em6.ControlNodes".cm.softCam.mendrelCathodeFrontAxisZ.up.inPos )
      Contact( "Unit1.Em6.ControlNodes".cm.softCam.mendrelCathodeFrontAxisY.backward.inPos )
   END_RUNG wire#w3
   RUNG wire#powerrail
      Contact( "Unit1.Em6.ControlNodes".cm.softCam.mendrelCathodeRearAxisZ.down.inPos )
   END_RUNG wire#w4
   RUNG wire#powerrail
      Contact( "Unit1.Em6.ControlNodes".cm.softCam.mendrelCathodeRearAxisZ.up.inPos )
      Contact( "Unit1.Em6.ControlNodes".cm.softCam.mendrelCathodeRearAxisY.backward.inPos )
   END_RUNG wire#w4
   RUNG wire#powerrail
      I_Contact( "Unit1.Em6.ControlNodes".stackTable."step".action1[183] )
      Not()
      Contact( "Unit1.Em6.ControlNodes".cm.Interlock.finalRollerRearAxisX.source.posAbsolute[0] )
      Move(in := 0, out1 => "Unit1.Em6.ControlNodes".cmFinalRollerRearAxisX.commands.selectSetPosition)
      Coil( "Unit1.Em6.ControlNodes".cm.Command.finalRollerRearAxisX.posAbsolute[0] )
   END_RUNG
   // the same network as SCL:
   #instFinalRollerRearAxisX_Position[0](PosiNo := 0,   // "Position.LER_Axis"
                           Status := #unitStatus,
                           int1 := "Unit1.Em6.ControlNodes".emRelations.em5.softCam.cathodeMainPnP2AxisX.alignTablePos.inPos,
                           int2 := "Unit1.Em6.ControlNodes".cm.softCam.mendrelAnodeFrontAxisZ.down.inPos OR ("Unit1.Em6.ControlNodes".cm.softCam.mendrelAnodeFrontAxisZ.up.inPos AND "Unit1.Em6.ControlNodes".cm.softCam.mendrelAnodeFrontAxisY.backward.inPos),
                           int3 := "Unit1.Em6.ControlNodes".cm.softCam.mendrelAnodeRearAxisZ.down.inPos OR ("Unit1.Em6.ControlNodes".cm.softCam.mendrelAnodeRearAxisZ.up.inPos AND "Unit1.Em6.ControlNodes".cm.softCam.mendrelAnodeRearAxisY.backward.inPos),
                           int4 := "Unit1.Em6.ControlNodes".cm.softCam.mendrelCathodeFrontAxisZ.down.inPos OR ("Unit1.Em6.ControlNodes".cm.softCam.mendrelCathodeFrontAxisZ.up.inPos AND "Unit1.Em6.ControlNodes".cm.softCam.mendrelCathodeFrontAxisY.backward.inPos),
                           int5 := "Unit1.Em6.ControlNodes".cm.softCam.mendrelCathodeRearAxisZ.down.inPos OR ("Unit1.Em6.ControlNodes".cm.softCam.mendrelCathodeRearAxisZ.up.inPos AND "Unit1.Em6.ControlNodes".cm.softCam.mendrelCathodeRearAxisY.backward.inPos),
                           commands := "Unit1.Em6.HmiInterface".cmFinalRollerRearAxisX.commands,
                           interlockOk := "Unit1.Em6.ControlNodes".cm.Interlock.finalRollerRearAxisX.source.posAbsolute,
                           intOut := "Unit1.Em6.HmiInterface".intCondition.Axis_22.Jog.intOut);
   #_w1 := NOT (NOT "Unit1.Em6.ControlNodes".stackTable."step".action1[183]) AND "Unit1.Em6.ControlNodes".cm.Interlock.finalRollerRearAxisX.source.posAbsolute[0];
   IF #_w1 THEN "Unit1.Em6.ControlNodes".cmFinalRollerRearAxisX.commands.selectSetPosition := 0; END_IF;
   "Unit1.Em6.ControlNodes".cm.Command.finalRollerRearAxisX.posAbsolute[0] := #_w1;
END_REGION

REGION Network 98: CmFinalRollerRearAxisX Position Absolute Position1
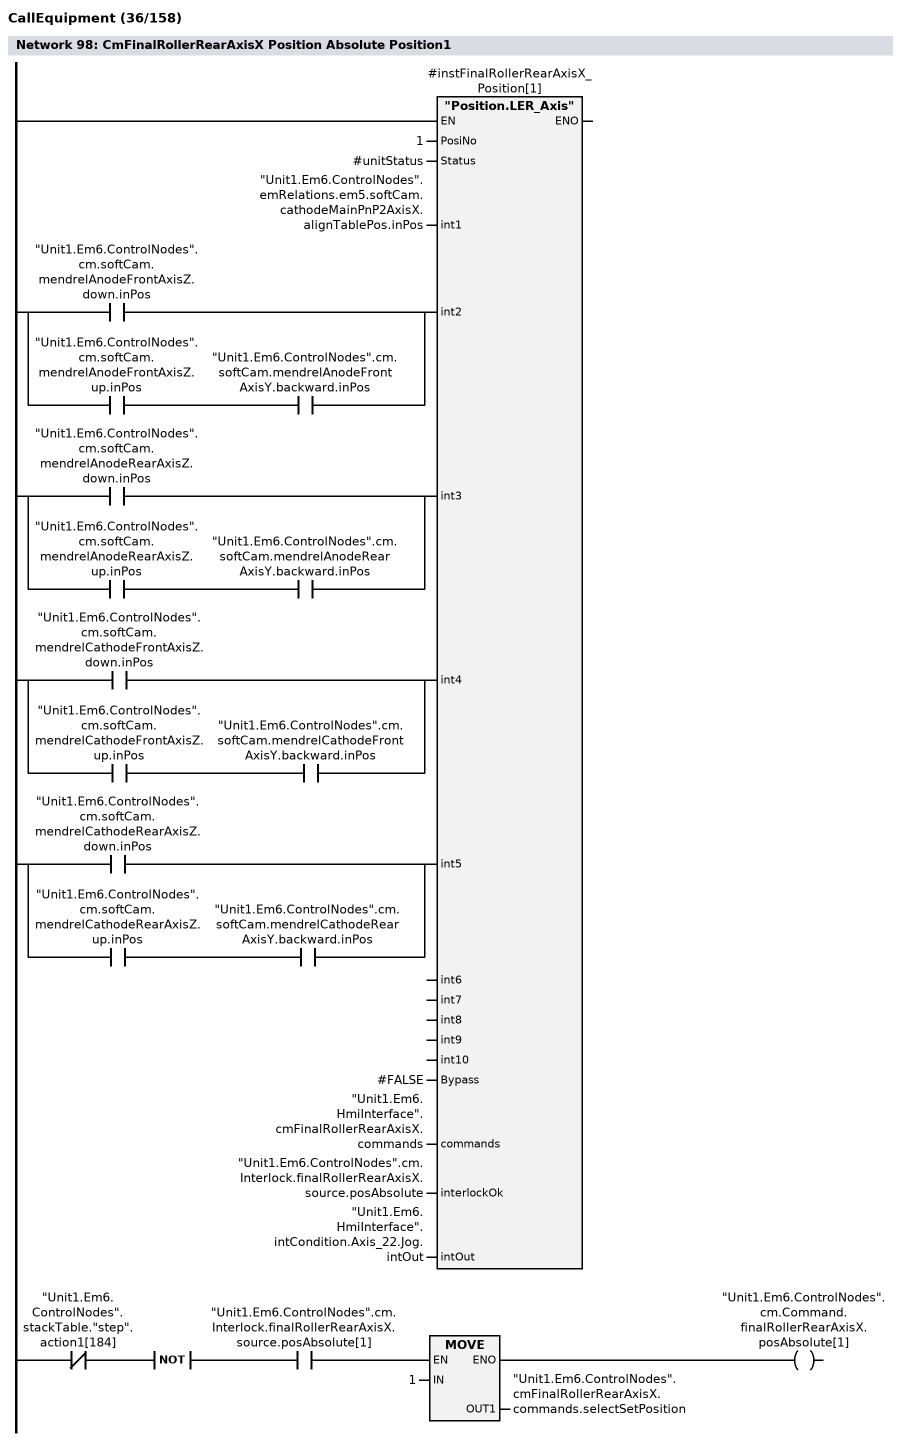
   RUNG wire#powerrail
      #instFinalRollerRearAxisX_Position[1](int2 := wire#w1, int3 := wire#w2, int4 := wire#w3, int5 := wire#w4, PosiNo := 1, Status := #unitStatus, int1 := "Unit1.Em6.ControlNodes".emRelations.em5.softCam.cathodeMainPnP2AxisX.alignTablePos.inPos, int6 :=, int7 :=, int8 :=, int9 :=, int10 :=, Bypass := #FALSE, commands := "Unit1.Em6.HmiInterface".cmFinalRollerRearAxisX.commands, interlockOk := "Unit1.Em6.ControlNodes".cm.Interlock.finalRollerRearAxisX.source.posAbsolute, intOut := "Unit1.Em6.HmiInterface".intCondition.Axis_22.Jog.intOut)
   END_RUNG
   RUNG wire#powerrail
      Contact( "Unit1.Em6.ControlNodes".cm.softCam.mendrelAnodeFrontAxisZ.down.inPos )
   END_RUNG wire#w1
   RUNG wire#powerrail
      Contact( "Unit1.Em6.ControlNodes".cm.softCam.mendrelAnodeFrontAxisZ.up.inPos )
      Contact( "Unit1.Em6.ControlNodes".cm.softCam.mendrelAnodeFrontAxisY.backward.inPos )
   END_RUNG wire#w1
   RUNG wire#powerrail
      Contact( "Unit1.Em6.ControlNodes".cm.softCam.mendrelAnodeRearAxisZ.down.inPos )
   END_RUNG wire#w2
   RUNG wire#powerrail
      Contact( "Unit1.Em6.ControlNodes".cm.softCam.mendrelAnodeRearAxisZ.up.inPos )
      Contact( "Unit1.Em6.ControlNodes".cm.softCam.mendrelAnodeRearAxisY.backward.inPos )
   END_RUNG wire#w2
   RUNG wire#powerrail
      Contact( "Unit1.Em6.ControlNodes".cm.softCam.mendrelCathodeFrontAxisZ.down.inPos )
   END_RUNG wire#w3
   RUNG wire#powerrail
      Contact( "Unit1.Em6.ControlNodes".cm.softCam.mendrelCathodeFrontAxisZ.up.inPos )
      Contact( "Unit1.Em6.ControlNodes".cm.softCam.mendrelCathodeFrontAxisY.backward.inPos )
   END_RUNG wire#w3
   RUNG wire#powerrail
      Contact( "Unit1.Em6.ControlNodes".cm.softCam.mendrelCathodeRearAxisZ.down.inPos )
   END_RUNG wire#w4
   RUNG wire#powerrail
      Contact( "Unit1.Em6.ControlNodes".cm.softCam.mendrelCathodeRearAxisZ.up.inPos )
      Contact( "Unit1.Em6.ControlNodes".cm.softCam.mendrelCathodeRearAxisY.backward.inPos )
   END_RUNG wire#w4
   RUNG wire#powerrail
      I_Contact( "Unit1.Em6.ControlNodes".stackTable."step".action1[184] )
      Not()
      Contact( "Unit1.Em6.ControlNodes".cm.Interlock.finalRollerRearAxisX.source.posAbsolute[1] )
      Move(in := 1, out1 => "Unit1.Em6.ControlNodes".cmFinalRollerRearAxisX.commands.selectSetPosition)
      Coil( "Unit1.Em6.ControlNodes".cm.Command.finalRollerRearAxisX.posAbsolute[1] )
   END_RUNG
   // the same network as SCL:
   #instFinalRollerRearAxisX_Position[1](PosiNo := 1,   // "Position.LER_Axis"
                           Status := #unitStatus,
                           int1 := "Unit1.Em6.ControlNodes".emRelations.em5.softCam.cathodeMainPnP2AxisX.alignTablePos.inPos,
                           int2 := "Unit1.Em6.ControlNodes".cm.softCam.mendrelAnodeFrontAxisZ.down.inPos OR ("Unit1.Em6.ControlNodes".cm.softCam.mendrelAnodeFrontAxisZ.up.inPos AND "Unit1.Em6.ControlNodes".cm.softCam.mendrelAnodeFrontAxisY.backward.inPos),
                           int3 := "Unit1.Em6.ControlNodes".cm.softCam.mendrelAnodeRearAxisZ.down.inPos OR ("Unit1.Em6.ControlNodes".cm.softCam.mendrelAnodeRearAxisZ.up.inPos AND "Unit1.Em6.ControlNodes".cm.softCam.mendrelAnodeRearAxisY.backward.inPos),
                           int4 := "Unit1.Em6.ControlNodes".cm.softCam.mendrelCathodeFrontAxisZ.down.inPos OR ("Unit1.Em6.ControlNodes".cm.softCam.mendrelCathodeFrontAxisZ.up.inPos AND "Unit1.Em6.ControlNodes".cm.softCam.mendrelCathodeFrontAxisY.backward.inPos),
                           int5 := "Unit1.Em6.ControlNodes".cm.softCam.mendrelCathodeRearAxisZ.down.inPos OR ("Unit1.Em6.ControlNodes".cm.softCam.mendrelCathodeRearAxisZ.up.inPos AND "Unit1.Em6.ControlNodes".cm.softCam.mendrelCathodeRearAxisY.backward.inPos),
                           Bypass := #FALSE,
                           commands := "Unit1.Em6.HmiInterface".cmFinalRollerRearAxisX.commands,
                           interlockOk := "Unit1.Em6.ControlNodes".cm.Interlock.finalRollerRearAxisX.source.posAbsolute,
                           intOut := "Unit1.Em6.HmiInterface".intCondition.Axis_22.Jog.intOut);
   #_w1 := NOT (NOT "Unit1.Em6.ControlNodes".stackTable."step".action1[184]) AND "Unit1.Em6.ControlNodes".cm.Interlock.finalRollerRearAxisX.source.posAbsolute[1];
   IF #_w1 THEN "Unit1.Em6.ControlNodes".cmFinalRollerRearAxisX.commands.selectSetPosition := 1; END_IF;
   "Unit1.Em6.ControlNodes".cm.Command.finalRollerRearAxisX.posAbsolute[1] := #_w1;
END_REGION

REGION Network 99: CmFinalRollerRearAxisX Position Absolute Position2
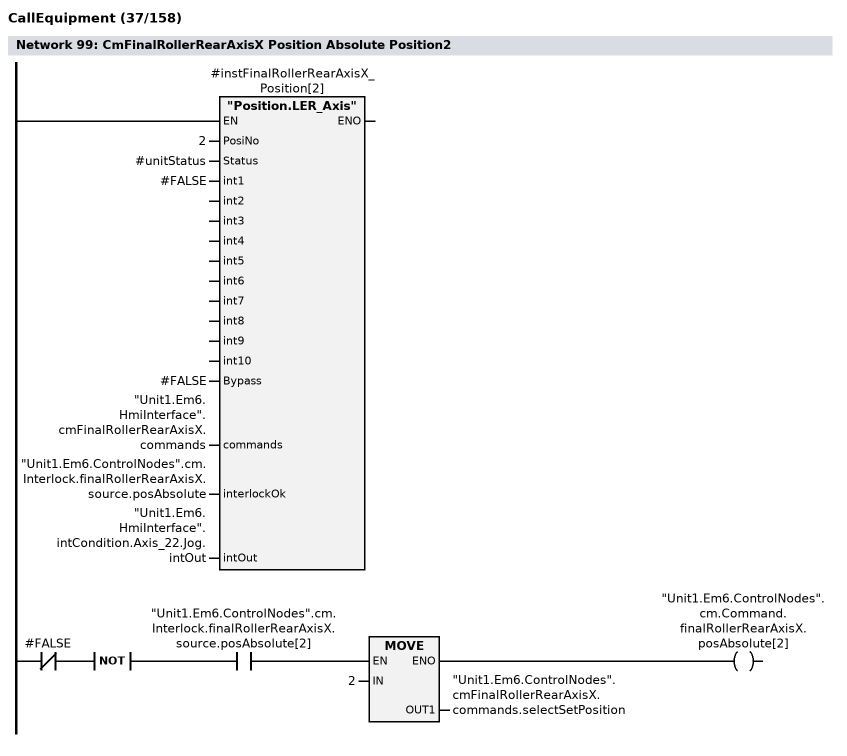
   RUNG wire#powerrail
      #instFinalRollerRearAxisX_Position[2](PosiNo := 2, Status := #unitStatus, int1 := #FALSE, int2 :=, int3 :=, int4 :=, int5 :=, int6 :=, int7 :=, int8 :=, int9 :=, int10 :=, Bypass := #FALSE, commands := "Unit1.Em6.HmiInterface".cmFinalRollerRearAxisX.commands, interlockOk := "Unit1.Em6.ControlNodes".cm.Interlock.finalRollerRearAxisX.source.posAbsolute, intOut := "Unit1.Em6.HmiInterface".intCondition.Axis_22.Jog.intOut)
   END_RUNG
   RUNG wire#powerrail
      I_Contact( #FALSE )
      Not()
      Contact( "Unit1.Em6.ControlNodes".cm.Interlock.finalRollerRearAxisX.source.posAbsolute[2] )
      Move(in := 2, out1 => "Unit1.Em6.ControlNodes".cmFinalRollerRearAxisX.commands.selectSetPosition)
      Coil( "Unit1.Em6.ControlNodes".cm.Command.finalRollerRearAxisX.posAbsolute[2] )
   END_RUNG
   // the same network as SCL:
   #instFinalRollerRearAxisX_Position[2](PosiNo := 2,   // "Position.LER_Axis"
                           Status := #unitStatus,
                           int1 := #FALSE,
                           Bypass := #FALSE,
                           commands := "Unit1.Em6.HmiInterface".cmFinalRollerRearAxisX.commands,
                           interlockOk := "Unit1.Em6.ControlNodes".cm.Interlock.finalRollerRearAxisX.source.posAbsolute,
                           intOut := "Unit1.Em6.HmiInterface".intCondition.Axis_22.Jog.intOut);
   #_w1 := NOT (NOT #FALSE) AND "Unit1.Em6.ControlNodes".cm.Interlock.finalRollerRearAxisX.source.posAbsolute[2];
   IF #_w1 THEN "Unit1.Em6.ControlNodes".cmFinalRollerRearAxisX.commands.selectSetPosition := 2; END_IF;
   "Unit1.Em6.ControlNodes".cm.Command.finalRollerRearAxisX.posAbsolute[2] := #_w1;
END_REGION

REGION Network 100: CmFinalRollerRearAxisX Position Absolute Position3
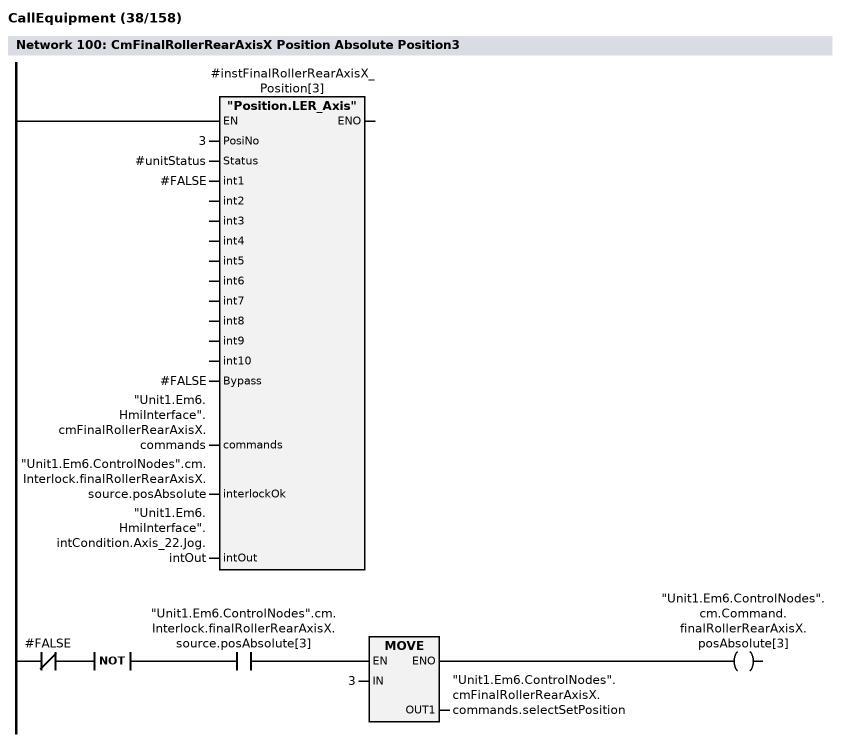
   RUNG wire#powerrail
      #instFinalRollerRearAxisX_Position[3](PosiNo := 3, Status := #unitStatus, int1 := #FALSE, int2 :=, int3 :=, int4 :=, int5 :=, int6 :=, int7 :=, int8 :=, int9 :=, int10 :=, Bypass := #FALSE, commands := "Unit1.Em6.HmiInterface".cmFinalRollerRearAxisX.commands, interlockOk := "Unit1.Em6.ControlNodes".cm.Interlock.finalRollerRearAxisX.source.posAbsolute, intOut := "Unit1.Em6.HmiInterface".intCondition.Axis_22.Jog.intOut)
   END_RUNG
   RUNG wire#powerrail
      I_Contact( #FALSE )
      Not()
      Contact( "Unit1.Em6.ControlNodes".cm.Interlock.finalRollerRearAxisX.source.posAbsolute[3] )
      Move(in := 3, out1 => "Unit1.Em6.ControlNodes".cmFinalRollerRearAxisX.commands.selectSetPosition)
      Coil( "Unit1.Em6.ControlNodes".cm.Command.finalRollerRearAxisX.posAbsolute[3] )
   END_RUNG
   // the same network as SCL:
   #instFinalRollerRearAxisX_Position[3](PosiNo := 3,   // "Position.LER_Axis"
                           Status := #unitStatus,
                           int1 := #FALSE,
                           Bypass := #FALSE,
                           commands := "Unit1.Em6.HmiInterface".cmFinalRollerRearAxisX.commands,
                           interlockOk := "Unit1.Em6.ControlNodes".cm.Interlock.finalRollerRearAxisX.source.posAbsolute,
                           intOut := "Unit1.Em6.HmiInterface".intCondition.Axis_22.Jog.intOut);
   #_w1 := NOT (NOT #FALSE) AND "Unit1.Em6.ControlNodes".cm.Interlock.finalRollerRearAxisX.source.posAbsolute[3];
   IF #_w1 THEN "Unit1.Em6.ControlNodes".cmFinalRollerRearAxisX.commands.selectSetPosition := 3; END_IF;
   "Unit1.Em6.ControlNodes".cm.Command.finalRollerRearAxisX.posAbsolute[3] := #_w1;
END_REGION

REGION Network 101: CmFinalRollerRearAxisX Position Absolute Position4
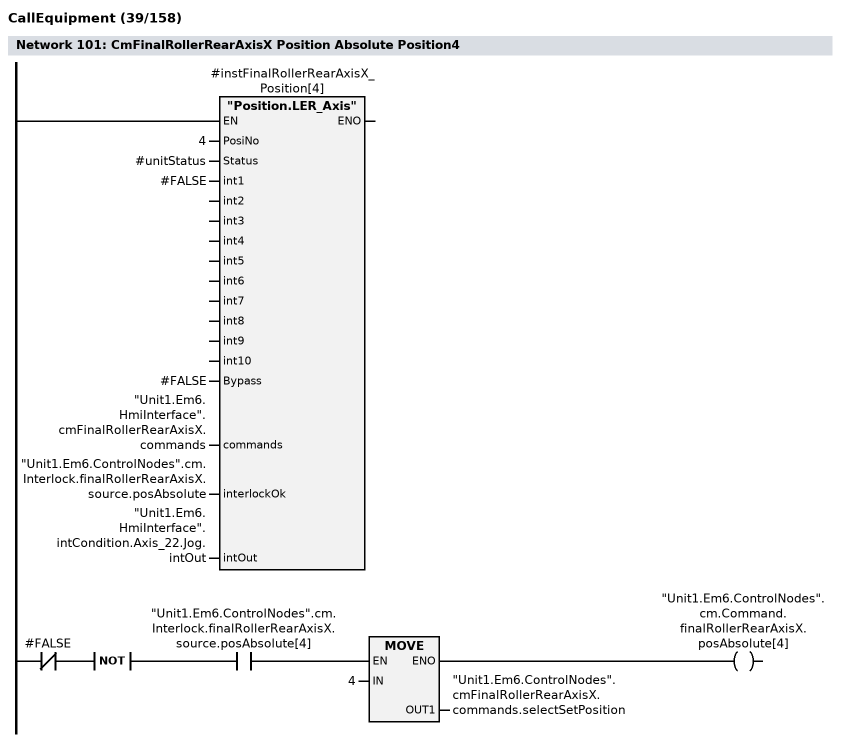
   RUNG wire#powerrail
      #instFinalRollerRearAxisX_Position[4](PosiNo := 4, Status := #unitStatus, int1 := #FALSE, int2 :=, int3 :=, int4 :=, int5 :=, int6 :=, int7 :=, int8 :=, int9 :=, int10 :=, Bypass := #FALSE, commands := "Unit1.Em6.HmiInterface".cmFinalRollerRearAxisX.commands, interlockOk := "Unit1.Em6.ControlNodes".cm.Interlock.finalRollerRearAxisX.source.posAbsolute, intOut := "Unit1.Em6.HmiInterface".intCondition.Axis_22.Jog.intOut)
   END_RUNG
   RUNG wire#powerrail
      I_Contact( #FALSE )
      Not()
      Contact( "Unit1.Em6.ControlNodes".cm.Interlock.finalRollerRearAxisX.source.posAbsolute[4] )
      Move(in := 4, out1 => "Unit1.Em6.ControlNodes".cmFinalRollerRearAxisX.commands.selectSetPosition)
      Coil( "Unit1.Em6.ControlNodes".cm.Command.finalRollerRearAxisX.posAbsolute[4] )
   END_RUNG
   // the same network as SCL:
   #instFinalRollerRearAxisX_Position[4](PosiNo := 4,   // "Position.LER_Axis"
                           Status := #unitStatus,
                           int1 := #FALSE,
                           Bypass := #FALSE,
                           commands := "Unit1.Em6.HmiInterface".cmFinalRollerRearAxisX.commands,
                           interlockOk := "Unit1.Em6.ControlNodes".cm.Interlock.finalRollerRearAxisX.source.posAbsolute,
                           intOut := "Unit1.Em6.HmiInterface".intCondition.Axis_22.Jog.intOut);
   #_w1 := NOT (NOT #FALSE) AND "Unit1.Em6.ControlNodes".cm.Interlock.finalRollerRearAxisX.source.posAbsolute[4];
   IF #_w1 THEN "Unit1.Em6.ControlNodes".cmFinalRollerRearAxisX.commands.selectSetPosition := 4; END_IF;
   "Unit1.Em6.ControlNodes".cm.Command.finalRollerRearAxisX.posAbsolute[4] := #_w1;
END_REGION

REGION Network 102: CmFinalRollerRearAxisX Position Absolute Position5
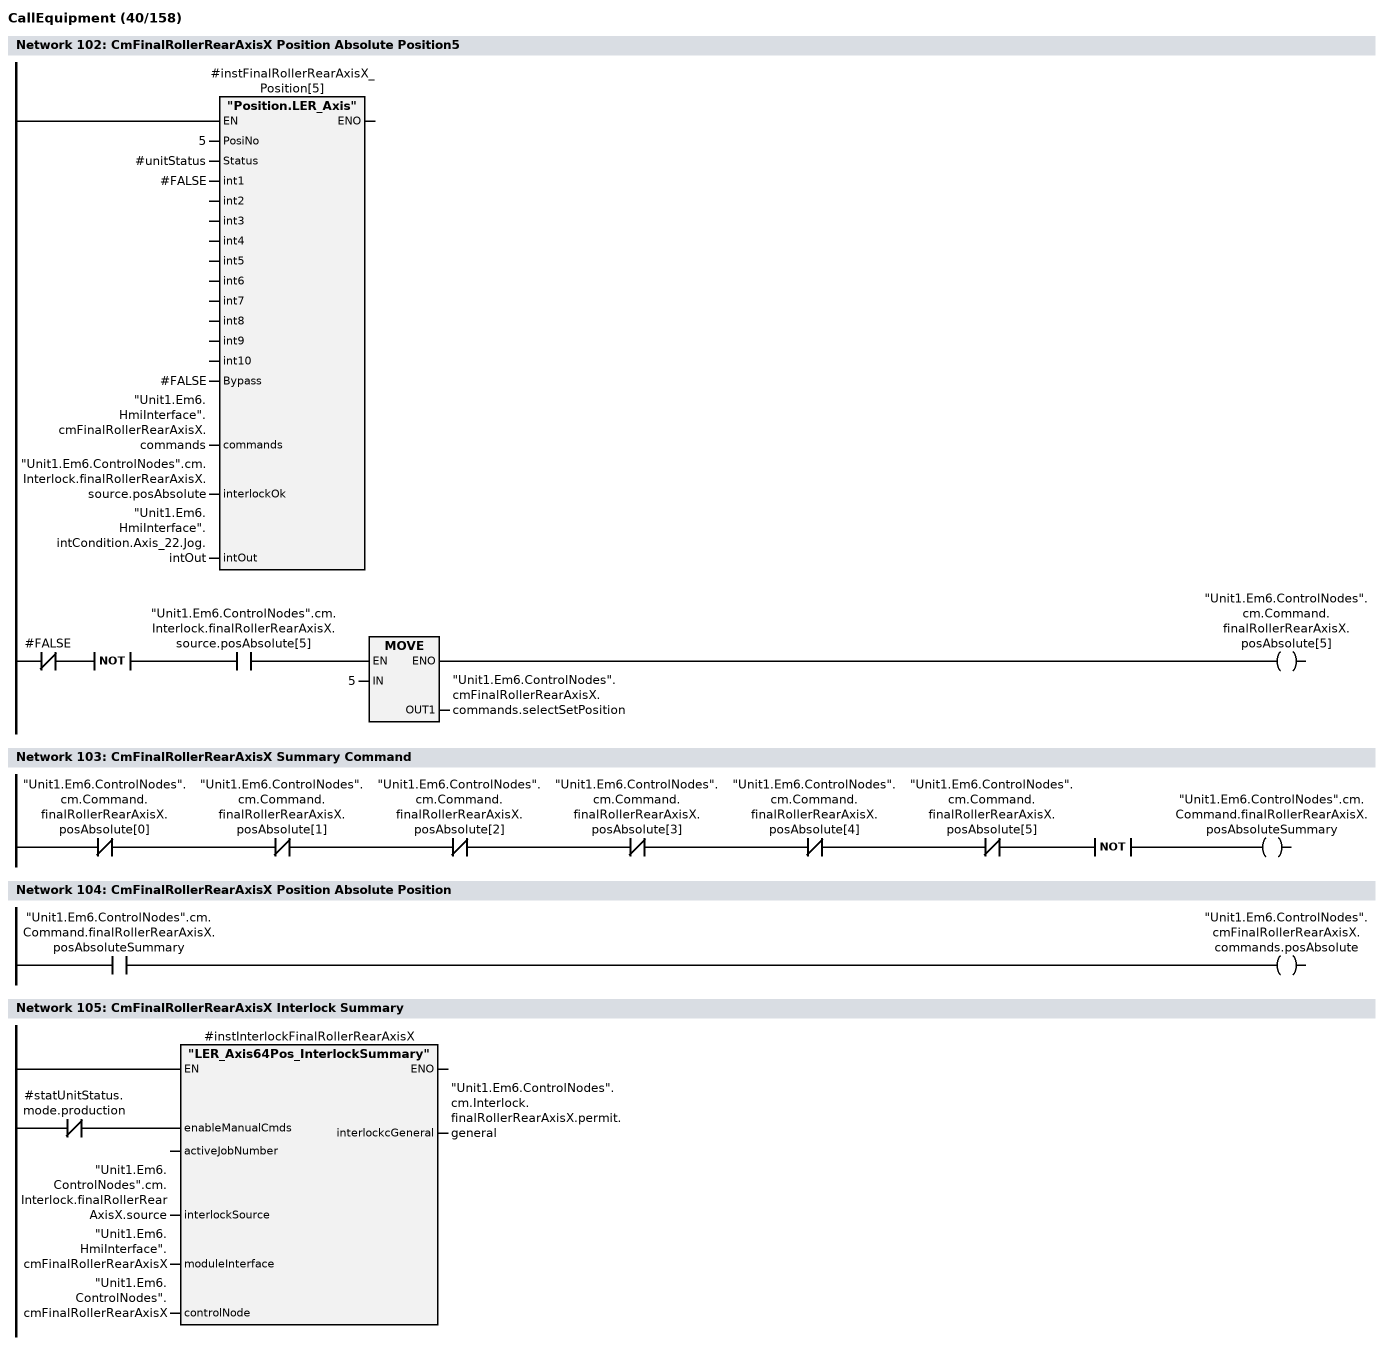
   RUNG wire#powerrail
      #instFinalRollerRearAxisX_Position[5](PosiNo := 5, Status := #unitStatus, int1 := #FALSE, int2 :=, int3 :=, int4 :=, int5 :=, int6 :=, int7 :=, int8 :=, int9 :=, int10 :=, Bypass := #FALSE, commands := "Unit1.Em6.HmiInterface".cmFinalRollerRearAxisX.commands, interlockOk := "Unit1.Em6.ControlNodes".cm.Interlock.finalRollerRearAxisX.source.posAbsolute, intOut := "Unit1.Em6.HmiInterface".intCondition.Axis_22.Jog.intOut)
   END_RUNG
   RUNG wire#powerrail
      I_Contact( #FALSE )
      Not()
      Contact( "Unit1.Em6.ControlNodes".cm.Interlock.finalRollerRearAxisX.source.posAbsolute[5] )
      Move(in := 5, out1 => "Unit1.Em6.ControlNodes".cmFinalRollerRearAxisX.commands.selectSetPosition)
      Coil( "Unit1.Em6.ControlNodes".cm.Command.finalRollerRearAxisX.posAbsolute[5] )
   END_RUNG
   // the same network as SCL:
   #instFinalRollerRearAxisX_Position[5](PosiNo := 5,   // "Position.LER_Axis"
                           Status := #unitStatus,
                           int1 := #FALSE,
                           Bypass := #FALSE,
                           commands := "Unit1.Em6.HmiInterface".cmFinalRollerRearAxisX.commands,
                           interlockOk := "Unit1.Em6.ControlNodes".cm.Interlock.finalRollerRearAxisX.source.posAbsolute,
                           intOut := "Unit1.Em6.HmiInterface".intCondition.Axis_22.Jog.intOut);
   #_w1 := NOT (NOT #FALSE) AND "Unit1.Em6.ControlNodes".cm.Interlock.finalRollerRearAxisX.source.posAbsolute[5];
   IF #_w1 THEN "Unit1.Em6.ControlNodes".cmFinalRollerRearAxisX.commands.selectSetPosition := 5; END_IF;
   "Unit1.Em6.ControlNodes".cm.Command.finalRollerRearAxisX.posAbsolute[5] := #_w1;
END_REGION

REGION Network 103: CmFinalRollerRearAxisX Summary Command
   RUNG wire#powerrail
      I_Contact( "Unit1.Em6.ControlNodes".cm.Command.finalRollerRearAxisX.posAbsolute[0] )
      I_Contact( "Unit1.Em6.ControlNodes".cm.Command.finalRollerRearAxisX.posAbsolute[1] )
      I_Contact( "Unit1.Em6.ControlNodes".cm.Command.finalRollerRearAxisX.posAbsolute[2] )
      I_Contact( "Unit1.Em6.ControlNodes".cm.Command.finalRollerRearAxisX.posAbsolute[3] )
      I_Contact( "Unit1.Em6.ControlNodes".cm.Command.finalRollerRearAxisX.posAbsolute[4] )
      I_Contact( "Unit1.Em6.ControlNodes".cm.Command.finalRollerRearAxisX.posAbsolute[5] )
      Not()
      Coil( "Unit1.Em6.ControlNodes".cm.Command.finalRollerRearAxisX.posAbsoluteSummary )
   END_RUNG
   // the same network as SCL:
   "Unit1.Em6.ControlNodes".cm.Command.finalRollerRearAxisX.posAbsoluteSummary := NOT (NOT "Unit1.Em6.ControlNodes".cm.Command.finalRollerRearAxisX.posAbsolute[0] AND NOT "Unit1.Em6.ControlNodes".cm.Command.finalRollerRearAxisX.posAbsolute[1] AND NOT "Unit1.Em6.ControlNodes".cm.Command.finalRollerRearAxisX.posAbsolute[2] AND NOT "Unit1.Em6.ControlNodes".cm.Command.finalRollerRearAxisX.posAbsolute[3] AND NOT "Unit1.Em6.ControlNodes".cm.Command.finalRollerRearAxisX.posAbsolute[4] AND NOT "Unit1.Em6.ControlNodes".cm.Command.finalRollerRearAxisX.posAbsolute[5]);
END_REGION

REGION Network 104: CmFinalRollerRearAxisX Position Absolute Position
   RUNG wire#powerrail
      Contact( "Unit1.Em6.ControlNodes".cm.Command.finalRollerRearAxisX.posAbsoluteSummary )
      Coil( "Unit1.Em6.ControlNodes".cmFinalRollerRearAxisX.commands.posAbsolute )
   END_RUNG
   // the same network as SCL:
   "Unit1.Em6.ControlNodes".cmFinalRollerRearAxisX.commands.posAbsolute := "Unit1.Em6.ControlNodes".cm.Command.finalRollerRearAxisX.posAbsoluteSummary;
END_REGION

REGION Network 105: CmFinalRollerRearAxisX Interlock Summary
   RUNG wire#powerrail
      #instInterlockFinalRollerRearAxisX(enableManualCmds := wire#w1, activeJobNumber :=, interlockSource := "Unit1.Em6.ControlNodes".cm.Interlock.finalRollerRearAxisX.source, moduleInterface := "Unit1.Em6.HmiInterface".cmFinalRollerRearAxisX, controlNode := "Unit1.Em6.ControlNodes".cmFinalRollerRearAxisX, interlockcGeneral => "Unit1.Em6.ControlNodes".cm.Interlock.finalRollerRearAxisX.permit.general)
   END_RUNG
   RUNG wire#powerrail
      I_Contact( #statUnitStatus.mode.production )
   END_RUNG wire#w1
   // the same network as SCL:
   #instInterlockFinalRollerRearAxisX(enableManualCmds := NOT #statUnitStatus.mode.production,   // "LER_Axis64Pos_InterlockSummary"
                           interlockSource := "Unit1.Em6.ControlNodes".cm.Interlock.finalRollerRearAxisX.source,
                           moduleInterface := "Unit1.Em6.HmiInterface".cmFinalRollerRearAxisX,
                           controlNode := "Unit1.Em6.ControlNodes".cmFinalRollerRearAxisX,
                           interlockcGeneral => "Unit1.Em6.ControlNodes".cm.Interlock.finalRollerRearAxisX.permit.general);
END_REGION

REGION Network 106: CmFinalRollerRearAxisX velocity/speed
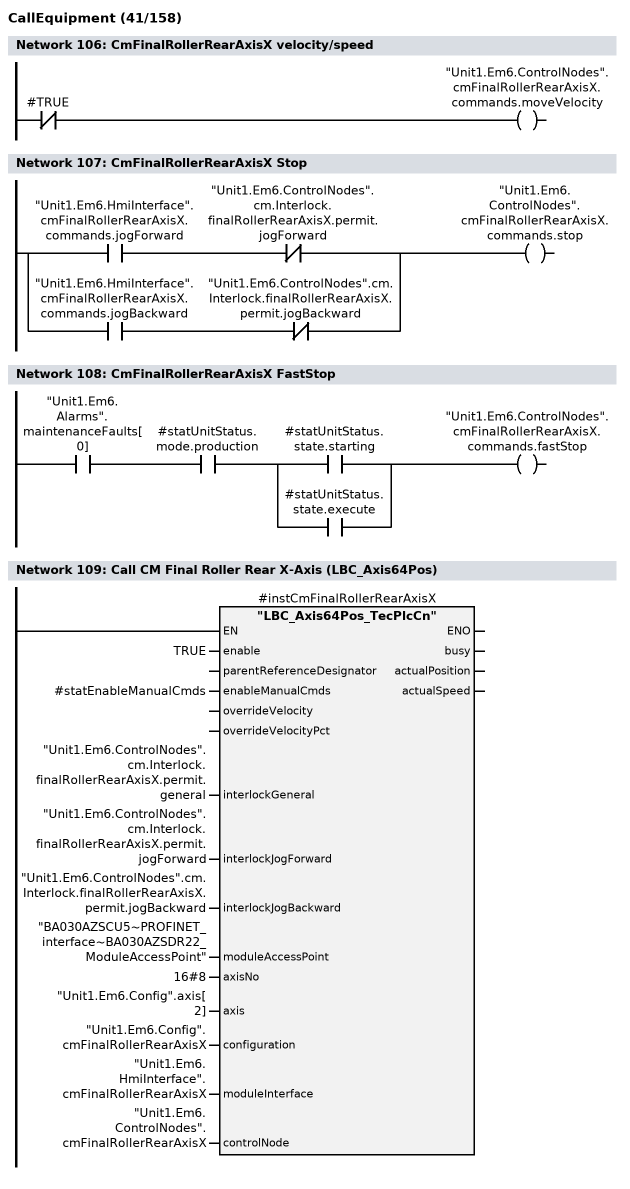
   RUNG wire#powerrail
      I_Contact( #TRUE )
      Coil( "Unit1.Em6.ControlNodes".cmFinalRollerRearAxisX.commands.moveVelocity )
   END_RUNG
   // the same network as SCL:
   "Unit1.Em6.ControlNodes".cmFinalRollerRearAxisX.commands.moveVelocity := NOT #TRUE;
END_REGION

REGION Network 107: CmFinalRollerRearAxisX Stop
   RUNG wire#powerrail
      Contact( "Unit1.Em6.HmiInterface".cmFinalRollerRearAxisX.commands.jogForward )
      I_Contact( "Unit1.Em6.ControlNodes".cm.Interlock.finalRollerRearAxisX.permit.jogForward )
      wire#w1
      Coil( "Unit1.Em6.ControlNodes".cmFinalRollerRearAxisX.commands.stop )
   END_RUNG
   RUNG wire#powerrail
      Contact( "Unit1.Em6.HmiInterface".cmFinalRollerRearAxisX.commands.jogBackward )
      I_Contact( "Unit1.Em6.ControlNodes".cm.Interlock.finalRollerRearAxisX.permit.jogBackward )
   END_RUNG wire#w1
   // the same network as SCL:
   "Unit1.Em6.ControlNodes".cmFinalRollerRearAxisX.commands.stop := ("Unit1.Em6.HmiInterface".cmFinalRollerRearAxisX.commands.jogForward AND NOT "Unit1.Em6.ControlNodes".cm.Interlock.finalRollerRearAxisX.permit.jogForward) OR ("Unit1.Em6.HmiInterface".cmFinalRollerRearAxisX.commands.jogBackward AND NOT "Unit1.Em6.ControlNodes".cm.Interlock.finalRollerRearAxisX.permit.jogBackward);
END_REGION

REGION Network 108: CmFinalRollerRearAxisX FastStop
   RUNG wire#powerrail
      Contact( "Unit1.Em6.Alarms".maintenanceFaults[0] )
      Contact( #statUnitStatus.mode.production )
      wire#w1
      Contact( #statUnitStatus.state.starting )
      wire#w2
      Coil( "Unit1.Em6.ControlNodes".cmFinalRollerRearAxisX.commands.fastStop )
   END_RUNG
   RUNG wire#w1
      Contact( #statUnitStatus.state.execute )
   END_RUNG wire#w2
   // the same network as SCL:
   "Unit1.Em6.ControlNodes".cmFinalRollerRearAxisX.commands.fastStop := "Unit1.Em6.Alarms".maintenanceFaults[0] AND #statUnitStatus.mode.production AND (#statUnitStatus.state.starting OR #statUnitStatus.state.execute);
END_REGION

REGION Network 109: Call CM Final Roller Rear X-Axis (LBC_Axis64Pos)
   RUNG wire#powerrail
      #instCmFinalRollerRearAxisX(enable := TRUE, parentReferenceDesignator :=, enableManualCmds := #statEnableManualCmds, overrideVelocity :=, overrideVelocityPct :=, interlockGeneral := "Unit1.Em6.ControlNodes".cm.Interlock.finalRollerRearAxisX.permit.general, interlockJogForward := "Unit1.Em6.ControlNodes".cm.Interlock.finalRollerRearAxisX.permit.jogForward, interlockJogBackward := "Unit1.Em6.ControlNodes".cm.Interlock.finalRollerRearAxisX.permit.jogBackward, moduleAccessPoint := "BA030AZSCU5~PROFINET_interface~BA030AZSDR22_ModuleAccessPoint", axisNo := 16#8, axis := "Unit1.Em6.Config".axis[2], configuration := "Unit1.Em6.Config".cmFinalRollerRearAxisX, moduleInterface := "Unit1.Em6.HmiInterface".cmFinalRollerRearAxisX, controlNode := "Unit1.Em6.ControlNodes".cmFinalRollerRearAxisX, busy =>, actualPosition =>, actualSpeed =>)
   END_RUNG
   // the same network as SCL:
   #instCmFinalRollerRearAxisX(enable := TRUE,   // "LBC_Axis64Pos_TecPlcCn"
                           enableManualCmds := #statEnableManualCmds,
                           interlockGeneral := "Unit1.Em6.ControlNodes".cm.Interlock.finalRollerRearAxisX.permit.general,
                           interlockJogForward := "Unit1.Em6.ControlNodes".cm.Interlock.finalRollerRearAxisX.permit.jogForward,
                           interlockJogBackward := "Unit1.Em6.ControlNodes".cm.Interlock.finalRollerRearAxisX.permit.jogBackward,
                           moduleAccessPoint := "BA030AZSCU5~PROFINET_interface~BA030AZSDR22_ModuleAccessPoint",
                           axisNo := 16#8,
                           axis := "Unit1.Em6.Config".axis[2],
                           configuration := "Unit1.Em6.Config".cmFinalRollerRearAxisX,
                           moduleInterface := "Unit1.Em6.HmiInterface".cmFinalRollerRearAxisX,
                           controlNode := "Unit1.Em6.ControlNodes".cmFinalRollerRearAxisX);
END_REGION

REGION Network 110: CmCathodeMainPnP1AxisX SoftCam
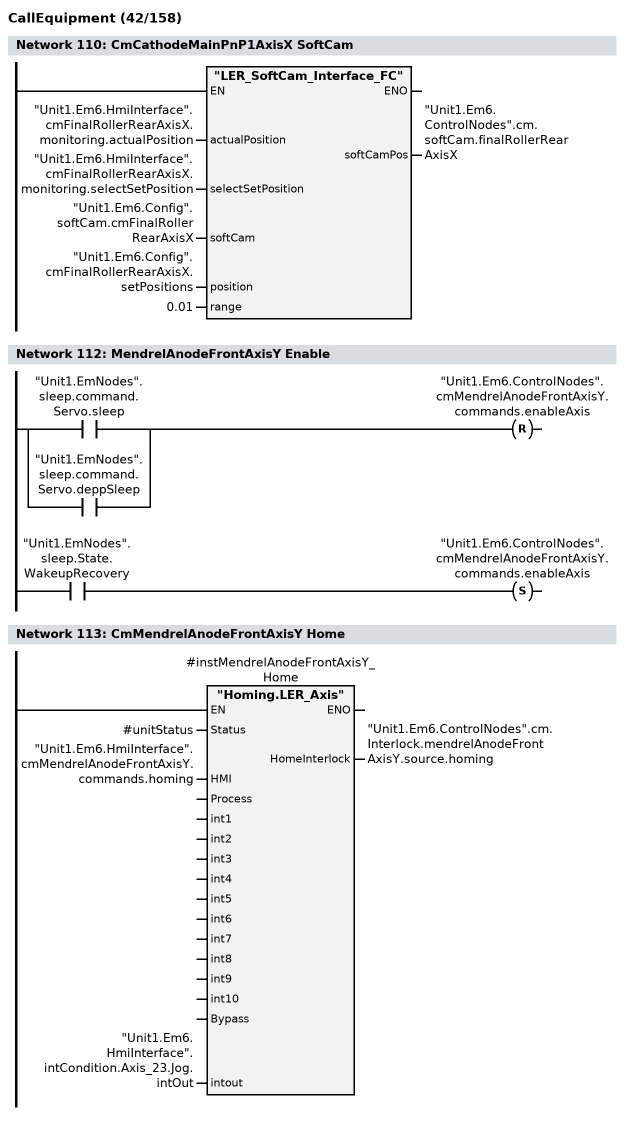
   RUNG wire#powerrail
      "LER_SoftCam_Interface_FC"(actualPosition := "Unit1.Em6.HmiInterface".cmFinalRollerRearAxisX.monitoring.actualPosition, selectSetPosition := "Unit1.Em6.HmiInterface".cmFinalRollerRearAxisX.monitoring.selectSetPosition, softCam := "Unit1.Em6.Config".softCam.cmFinalRollerRearAxisX, position := "Unit1.Em6.Config".cmFinalRollerRearAxisX.setPositions, range := 0.01, softCamPos => "Unit1.Em6.ControlNodes".cm.softCam.finalRollerRearAxisX)
   END_RUNG
   // the same network as SCL:
   "LER_SoftCam_Interface_FC"(actualPosition := "Unit1.Em6.HmiInterface".cmFinalRollerRearAxisX.monitoring.actualPosition,
                           selectSetPosition := "Unit1.Em6.HmiInterface".cmFinalRollerRearAxisX.monitoring.selectSetPosition,
                           softCam := "Unit1.Em6.Config".softCam.cmFinalRollerRearAxisX,
                           position := "Unit1.Em6.Config".cmFinalRollerRearAxisX.setPositions,
                           range := 0.01,
                           softCamPos => "Unit1.Em6.ControlNodes".cm.softCam.finalRollerRearAxisX);
END_REGION

REGION Network 112: MendrelAnodeFrontAxisY Enable
   RUNG wire#powerrail
      Contact( "Unit1.EmNodes".sleep.command.Servo.sleep )
      wire#w1
      R_Coil( "Unit1.Em6.ControlNodes".cmMendrelAnodeFrontAxisY.commands.enableAxis )
   END_RUNG
   RUNG wire#powerrail
      Contact( "Unit1.EmNodes".sleep.command.Servo.deppSleep )
   END_RUNG wire#w1
   RUNG wire#powerrail
      Contact( "Unit1.EmNodes".sleep.State.WakeupRecovery )
      S_Coil( "Unit1.Em6.ControlNodes".cmMendrelAnodeFrontAxisY.commands.enableAxis )
   END_RUNG
   // the same network as SCL:
   IF "Unit1.EmNodes".sleep.command.Servo.sleep OR "Unit1.EmNodes".sleep.command.Servo.deppSleep THEN
       "Unit1.Em6.ControlNodes".cmMendrelAnodeFrontAxisY.commands.enableAxis := FALSE;
   END_IF;
   IF "Unit1.EmNodes".sleep.State.WakeupRecovery THEN
       "Unit1.Em6.ControlNodes".cmMendrelAnodeFrontAxisY.commands.enableAxis := TRUE;
   END_IF;
END_REGION

REGION Network 113: CmMendrelAnodeFrontAxisY Home
   RUNG wire#powerrail
      #instMendrelAnodeFrontAxisY_Home(Status := #unitStatus, HMI := "Unit1.Em6.HmiInterface".cmMendrelAnodeFrontAxisY.commands.homing, Process :=, int1 :=, int2 :=, int3 :=, int4 :=, int5 :=, int6 :=, int7 :=, int8 :=, int9 :=, int10 :=, Bypass :=, intout := "Unit1.Em6.HmiInterface".intCondition.Axis_23.Jog.intOut, HomeInterlock => "Unit1.Em6.ControlNodes".cm.Interlock.mendrelAnodeFrontAxisY.source.homing)
   END_RUNG
   // the same network as SCL:
   #instMendrelAnodeFrontAxisY_Home(Status := #unitStatus,   // "Homing.LER_Axis"
                           HMI := "Unit1.Em6.HmiInterface".cmMendrelAnodeFrontAxisY.commands.homing,
                           intout := "Unit1.Em6.HmiInterface".intCondition.Axis_23.Jog.intOut,
                           HomeInterlock => "Unit1.Em6.ControlNodes".cm.Interlock.mendrelAnodeFrontAxisY.source.homing);
END_REGION

REGION Network 114: CmMendrelAnodeFrontAxisY Position Absolute Jog
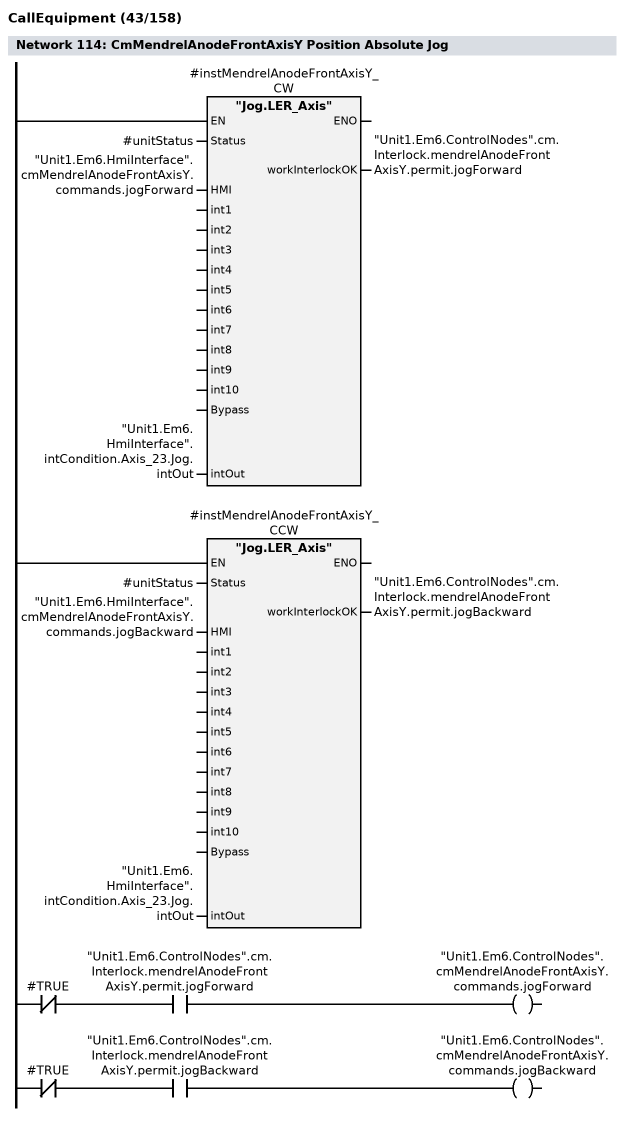
   RUNG wire#powerrail
      #instMendrelAnodeFrontAxisY_CW(Status := #unitStatus, HMI := "Unit1.Em6.HmiInterface".cmMendrelAnodeFrontAxisY.commands.jogForward, int1 :=, int2 :=, int3 :=, int4 :=, int5 :=, int6 :=, int7 :=, int8 :=, int9 :=, int10 :=, Bypass :=, intOut := "Unit1.Em6.HmiInterface".intCondition.Axis_23.Jog.intOut, workInterlockOK => "Unit1.Em6.ControlNodes".cm.Interlock.mendrelAnodeFrontAxisY.permit.jogForward)
   END_RUNG
   RUNG wire#powerrail
      #instMendrelAnodeFrontAxisY_CCW(Status := #unitStatus, HMI := "Unit1.Em6.HmiInterface".cmMendrelAnodeFrontAxisY.commands.jogBackward, int1 :=, int2 :=, int3 :=, int4 :=, int5 :=, int6 :=, int7 :=, int8 :=, int9 :=, int10 :=, Bypass :=, intOut := "Unit1.Em6.HmiInterface".intCondition.Axis_23.Jog.intOut, workInterlockOK => "Unit1.Em6.ControlNodes".cm.Interlock.mendrelAnodeFrontAxisY.permit.jogBackward)
   END_RUNG
   RUNG wire#powerrail
      I_Contact( #TRUE )
      Contact( "Unit1.Em6.ControlNodes".cm.Interlock.mendrelAnodeFrontAxisY.permit.jogForward )
      Coil( "Unit1.Em6.ControlNodes".cmMendrelAnodeFrontAxisY.commands.jogForward )
   END_RUNG
   RUNG wire#powerrail
      I_Contact( #TRUE )
      Contact( "Unit1.Em6.ControlNodes".cm.Interlock.mendrelAnodeFrontAxisY.permit.jogBackward )
      Coil( "Unit1.Em6.ControlNodes".cmMendrelAnodeFrontAxisY.commands.jogBackward )
   END_RUNG
   // the same network as SCL:
   #instMendrelAnodeFrontAxisY_CW(Status := #unitStatus,   // "Jog.LER_Axis"
                           HMI := "Unit1.Em6.HmiInterface".cmMendrelAnodeFrontAxisY.commands.jogForward,
                           intOut := "Unit1.Em6.HmiInterface".intCondition.Axis_23.Jog.intOut,
                           workInterlockOK => "Unit1.Em6.ControlNodes".cm.Interlock.mendrelAnodeFrontAxisY.permit.jogForward);
   #instMendrelAnodeFrontAxisY_CCW(Status := #unitStatus,   // "Jog.LER_Axis"
                           HMI := "Unit1.Em6.HmiInterface".cmMendrelAnodeFrontAxisY.commands.jogBackward,
                           intOut := "Unit1.Em6.HmiInterface".intCondition.Axis_23.Jog.intOut,
                           workInterlockOK => "Unit1.Em6.ControlNodes".cm.Interlock.mendrelAnodeFrontAxisY.permit.jogBackward);
   "Unit1.Em6.ControlNodes".cmMendrelAnodeFrontAxisY.commands.jogForward := NOT #TRUE AND "Unit1.Em6.ControlNodes".cm.Interlock.mendrelAnodeFrontAxisY.permit.jogForward;
   "Unit1.Em6.ControlNodes".cmMendrelAnodeFrontAxisY.commands.jogBackward := NOT #TRUE AND "Unit1.Em6.ControlNodes".cm.Interlock.mendrelAnodeFrontAxisY.permit.jogBackward;
END_REGION

REGION Network 115: CmMendrelAnodeFrontAxisY Position Absolute Position0
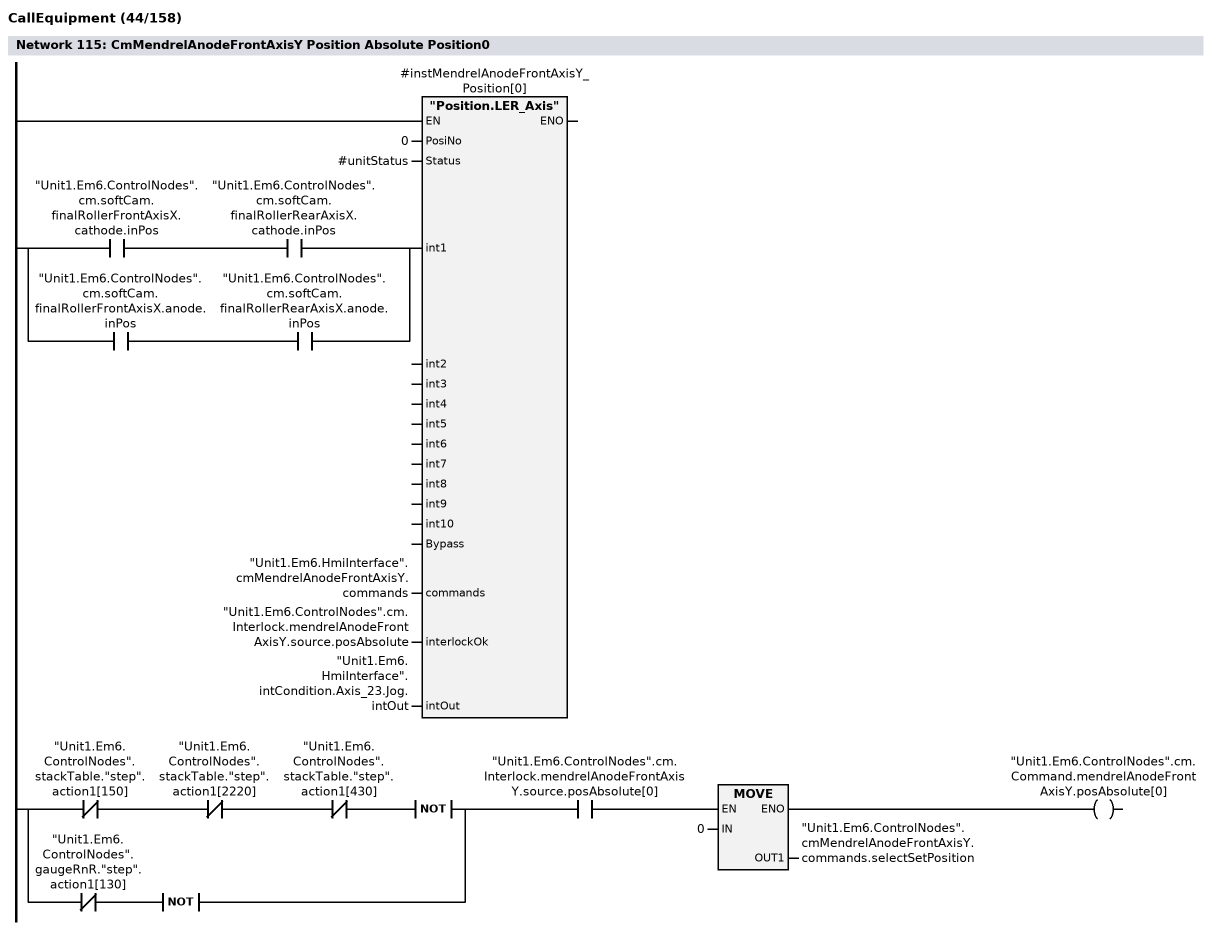
   RUNG wire#powerrail
      #instMendrelAnodeFrontAxisY_Position[0](int1 := wire#w1, PosiNo := 0, Status := #unitStatus, int2 :=, int3 :=, int4 :=, int5 :=, int6 :=, int7 :=, int8 :=, int9 :=, int10 :=, Bypass :=, commands := "Unit1.Em6.HmiInterface".cmMendrelAnodeFrontAxisY.commands, interlockOk := "Unit1.Em6.ControlNodes".cm.Interlock.mendrelAnodeFrontAxisY.source.posAbsolute, intOut := "Unit1.Em6.HmiInterface".intCondition.Axis_23.Jog.intOut)
   END_RUNG
   RUNG wire#powerrail
      Contact( "Unit1.Em6.ControlNodes".cm.softCam.finalRollerFrontAxisX.cathode.inPos )
      Contact( "Unit1.Em6.ControlNodes".cm.softCam.finalRollerRearAxisX.cathode.inPos )
   END_RUNG wire#w1
   RUNG wire#powerrail
      Contact( "Unit1.Em6.ControlNodes".cm.softCam.finalRollerFrontAxisX.anode.inPos )
      Contact( "Unit1.Em6.ControlNodes".cm.softCam.finalRollerRearAxisX.anode.inPos )
   END_RUNG wire#w1
   RUNG wire#powerrail
      I_Contact( "Unit1.Em6.ControlNodes".stackTable."step".action1[150] )
      I_Contact( "Unit1.Em6.ControlNodes".stackTable."step".action1[2220] )
      I_Contact( "Unit1.Em6.ControlNodes".stackTable."step".action1[430] )
      Not()
      wire#w2
      Contact( "Unit1.Em6.ControlNodes".cm.Interlock.mendrelAnodeFrontAxisY.source.posAbsolute[0] )
      Move(in := 0, out1 => "Unit1.Em6.ControlNodes".cmMendrelAnodeFrontAxisY.commands.selectSetPosition)
      Coil( "Unit1.Em6.ControlNodes".cm.Command.mendrelAnodeFrontAxisY.posAbsolute[0] )
   END_RUNG
   RUNG wire#powerrail
      I_Contact( "Unit1.Em6.ControlNodes".gaugeRnR."step".action1[130] )
      Not()
   END_RUNG wire#w2
   // the same network as SCL:
   #instMendrelAnodeFrontAxisY_Position[0](PosiNo := 0,   // "Position.LER_Axis"
                           Status := #unitStatus,
                           int1 := ("Unit1.Em6.ControlNodes".cm.softCam.finalRollerFrontAxisX.cathode.inPos AND "Unit1.Em6.ControlNodes".cm.softCam.finalRollerRearAxisX.cathode.inPos) OR ("Unit1.Em6.ControlNodes".cm.softCam.finalRollerFrontAxisX.anode.inPos AND "Unit1.Em6.ControlNodes".cm.softCam.finalRollerRearAxisX.anode.inPos),
                           commands := "Unit1.Em6.HmiInterface".cmMendrelAnodeFrontAxisY.commands,
                           interlockOk := "Unit1.Em6.ControlNodes".cm.Interlock.mendrelAnodeFrontAxisY.source.posAbsolute,
                           intOut := "Unit1.Em6.HmiInterface".intCondition.Axis_23.Jog.intOut);
   #_w1 := (NOT (NOT "Unit1.Em6.ControlNodes".stackTable."step".action1[150] AND NOT "Unit1.Em6.ControlNodes".stackTable."step".action1[2220] AND NOT "Unit1.Em6.ControlNodes".stackTable."step".action1[430]) OR NOT (NOT "Unit1.Em6.ControlNodes".gaugeRnR."step".action1[130])) AND "Unit1.Em6.ControlNodes".cm.Interlock.mendrelAnodeFrontAxisY.source.posAbsolute[0];
   IF #_w1 THEN "Unit1.Em6.ControlNodes".cmMendrelAnodeFrontAxisY.commands.selectSetPosition := 0; END_IF;
   "Unit1.Em6.ControlNodes".cm.Command.mendrelAnodeFrontAxisY.posAbsolute[0] := #_w1;
END_REGION

REGION Network 116: CmMendrelAnodeFrontAxisY Position Absolute Position1
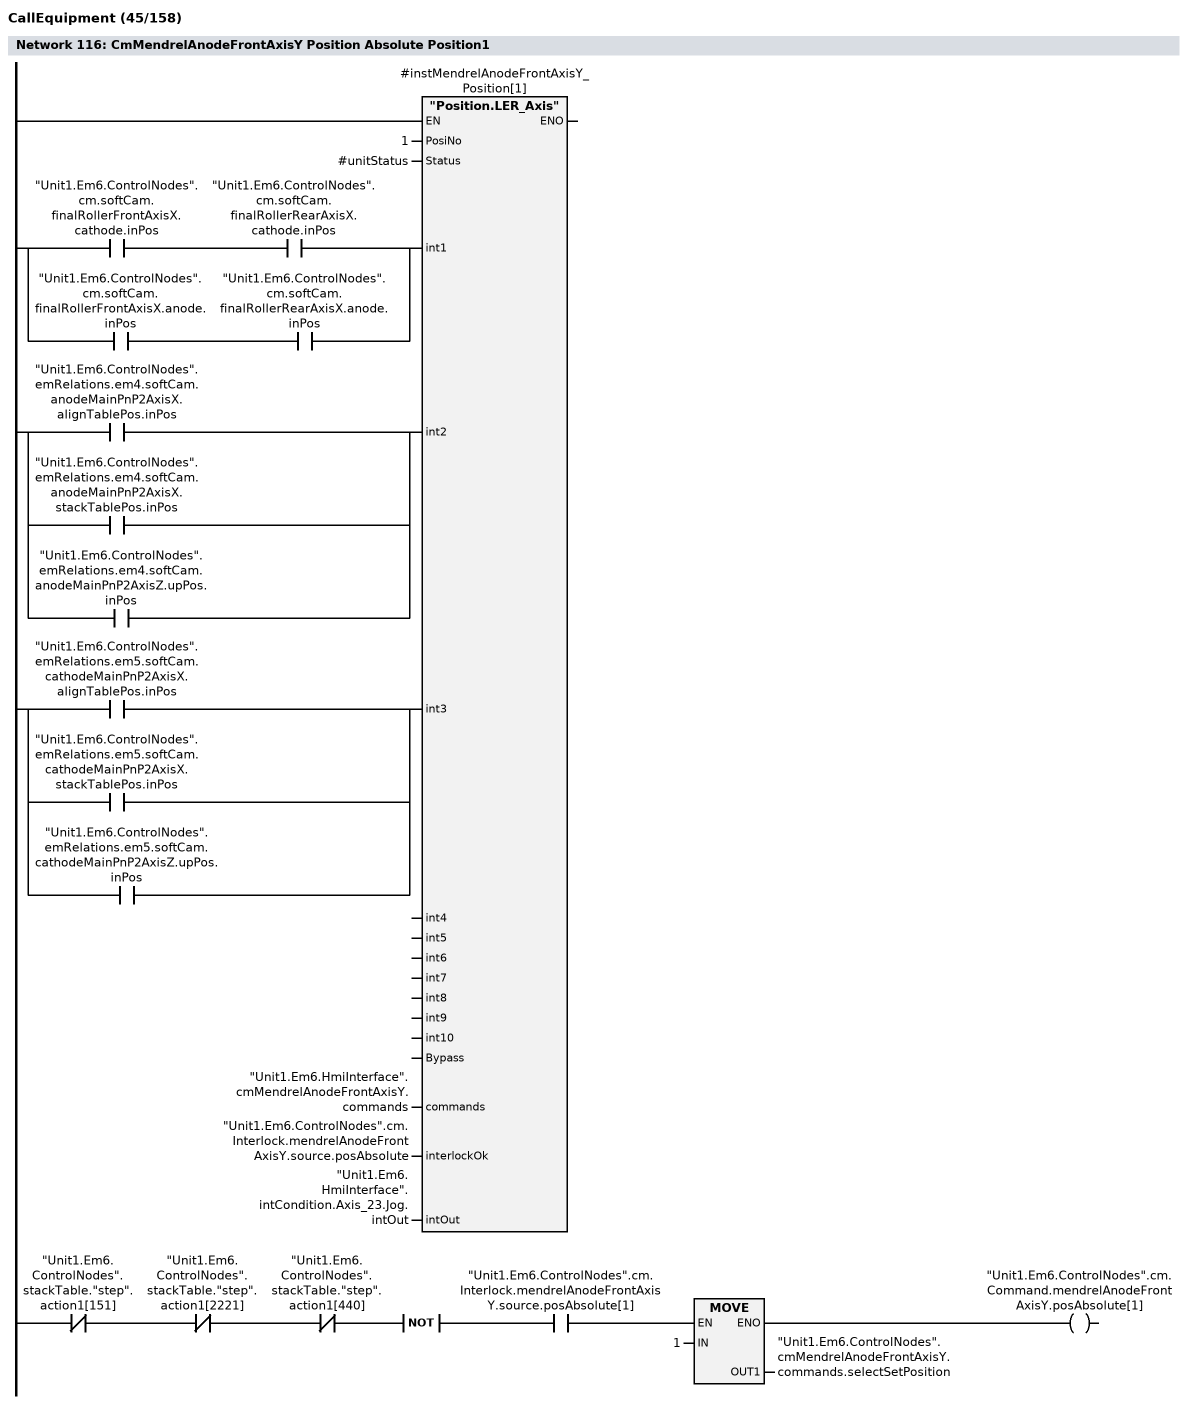
   RUNG wire#powerrail
      #instMendrelAnodeFrontAxisY_Position[1](int1 := wire#w1, int2 := wire#w2, int3 := wire#w3, PosiNo := 1, Status := #unitStatus, int4 :=, int5 :=, int6 :=, int7 :=, int8 :=, int9 :=, int10 :=, Bypass :=, commands := "Unit1.Em6.HmiInterface".cmMendrelAnodeFrontAxisY.commands, interlockOk := "Unit1.Em6.ControlNodes".cm.Interlock.mendrelAnodeFrontAxisY.source.posAbsolute, intOut := "Unit1.Em6.HmiInterface".intCondition.Axis_23.Jog.intOut)
   END_RUNG
   RUNG wire#powerrail
      Contact( "Unit1.Em6.ControlNodes".cm.softCam.finalRollerFrontAxisX.cathode.inPos )
      Contact( "Unit1.Em6.ControlNodes".cm.softCam.finalRollerRearAxisX.cathode.inPos )
   END_RUNG wire#w1
   RUNG wire#powerrail
      Contact( "Unit1.Em6.ControlNodes".cm.softCam.finalRollerFrontAxisX.anode.inPos )
      Contact( "Unit1.Em6.ControlNodes".cm.softCam.finalRollerRearAxisX.anode.inPos )
   END_RUNG wire#w1
   RUNG wire#powerrail
      Contact( "Unit1.Em6.ControlNodes".emRelations.em4.softCam.anodeMainPnP2AxisX.alignTablePos.inPos )
   END_RUNG wire#w2
   RUNG wire#powerrail
      Contact( "Unit1.Em6.ControlNodes".emRelations.em4.softCam.anodeMainPnP2AxisX.stackTablePos.inPos )
   END_RUNG wire#w2
   RUNG wire#powerrail
      Contact( "Unit1.Em6.ControlNodes".emRelations.em4.softCam.anodeMainPnP2AxisZ.upPos.inPos )
   END_RUNG wire#w2
   RUNG wire#powerrail
      Contact( "Unit1.Em6.ControlNodes".emRelations.em5.softCam.cathodeMainPnP2AxisX.alignTablePos.inPos )
   END_RUNG wire#w3
   RUNG wire#powerrail
      Contact( "Unit1.Em6.ControlNodes".emRelations.em5.softCam.cathodeMainPnP2AxisX.stackTablePos.inPos )
   END_RUNG wire#w3
   RUNG wire#powerrail
      Contact( "Unit1.Em6.ControlNodes".emRelations.em5.softCam.cathodeMainPnP2AxisZ.upPos.inPos )
   END_RUNG wire#w3
   RUNG wire#powerrail
      I_Contact( "Unit1.Em6.ControlNodes".stackTable."step".action1[151] )
      I_Contact( "Unit1.Em6.ControlNodes".stackTable."step".action1[2221] )
      I_Contact( "Unit1.Em6.ControlNodes".stackTable."step".action1[440] )
      Not()
      Contact( "Unit1.Em6.ControlNodes".cm.Interlock.mendrelAnodeFrontAxisY.source.posAbsolute[1] )
      Move(in := 1, out1 => "Unit1.Em6.ControlNodes".cmMendrelAnodeFrontAxisY.commands.selectSetPosition)
      Coil( "Unit1.Em6.ControlNodes".cm.Command.mendrelAnodeFrontAxisY.posAbsolute[1] )
   END_RUNG
   // the same network as SCL:
   #instMendrelAnodeFrontAxisY_Position[1](PosiNo := 1,   // "Position.LER_Axis"
                           Status := #unitStatus,
                           int1 := ("Unit1.Em6.ControlNodes".cm.softCam.finalRollerFrontAxisX.cathode.inPos AND "Unit1.Em6.ControlNodes".cm.softCam.finalRollerRearAxisX.cathode.inPos) OR ("Unit1.Em6.ControlNodes".cm.softCam.finalRollerFrontAxisX.anode.inPos AND "Unit1.Em6.ControlNodes".cm.softCam.finalRollerRearAxisX.anode.inPos),
                           int2 := "Unit1.Em6.ControlNodes".emRelations.em4.softCam.anodeMainPnP2AxisX.alignTablePos.inPos OR "Unit1.Em6.ControlNodes".emRelations.em4.softCam.anodeMainPnP2AxisX.stackTablePos.inPos OR "Unit1.Em6.ControlNodes".emRelations.em4.softCam.anodeMainPnP2AxisZ.upPos.inPos,
                           int3 := "Unit1.Em6.ControlNodes".emRelations.em5.softCam.cathodeMainPnP2AxisX.alignTablePos.inPos OR "Unit1.Em6.ControlNodes".emRelations.em5.softCam.cathodeMainPnP2AxisX.stackTablePos.inPos OR "Unit1.Em6.ControlNodes".emRelations.em5.softCam.cathodeMainPnP2AxisZ.upPos.inPos,
                           commands := "Unit1.Em6.HmiInterface".cmMendrelAnodeFrontAxisY.commands,
                           interlockOk := "Unit1.Em6.ControlNodes".cm.Interlock.mendrelAnodeFrontAxisY.source.posAbsolute,
                           intOut := "Unit1.Em6.HmiInterface".intCondition.Axis_23.Jog.intOut);
   #_w1 := NOT (NOT "Unit1.Em6.ControlNodes".stackTable."step".action1[151] AND NOT "Unit1.Em6.ControlNodes".stackTable."step".action1[2221] AND NOT "Unit1.Em6.ControlNodes".stackTable."step".action1[440]) AND "Unit1.Em6.ControlNodes".cm.Interlock.mendrelAnodeFrontAxisY.source.posAbsolute[1];
   IF #_w1 THEN "Unit1.Em6.ControlNodes".cmMendrelAnodeFrontAxisY.commands.selectSetPosition := 1; END_IF;
   "Unit1.Em6.ControlNodes".cm.Command.mendrelAnodeFrontAxisY.posAbsolute[1] := #_w1;
END_REGION

REGION Network 117: CmMendrelAnodeFrontAxisY Position Absolute Position2
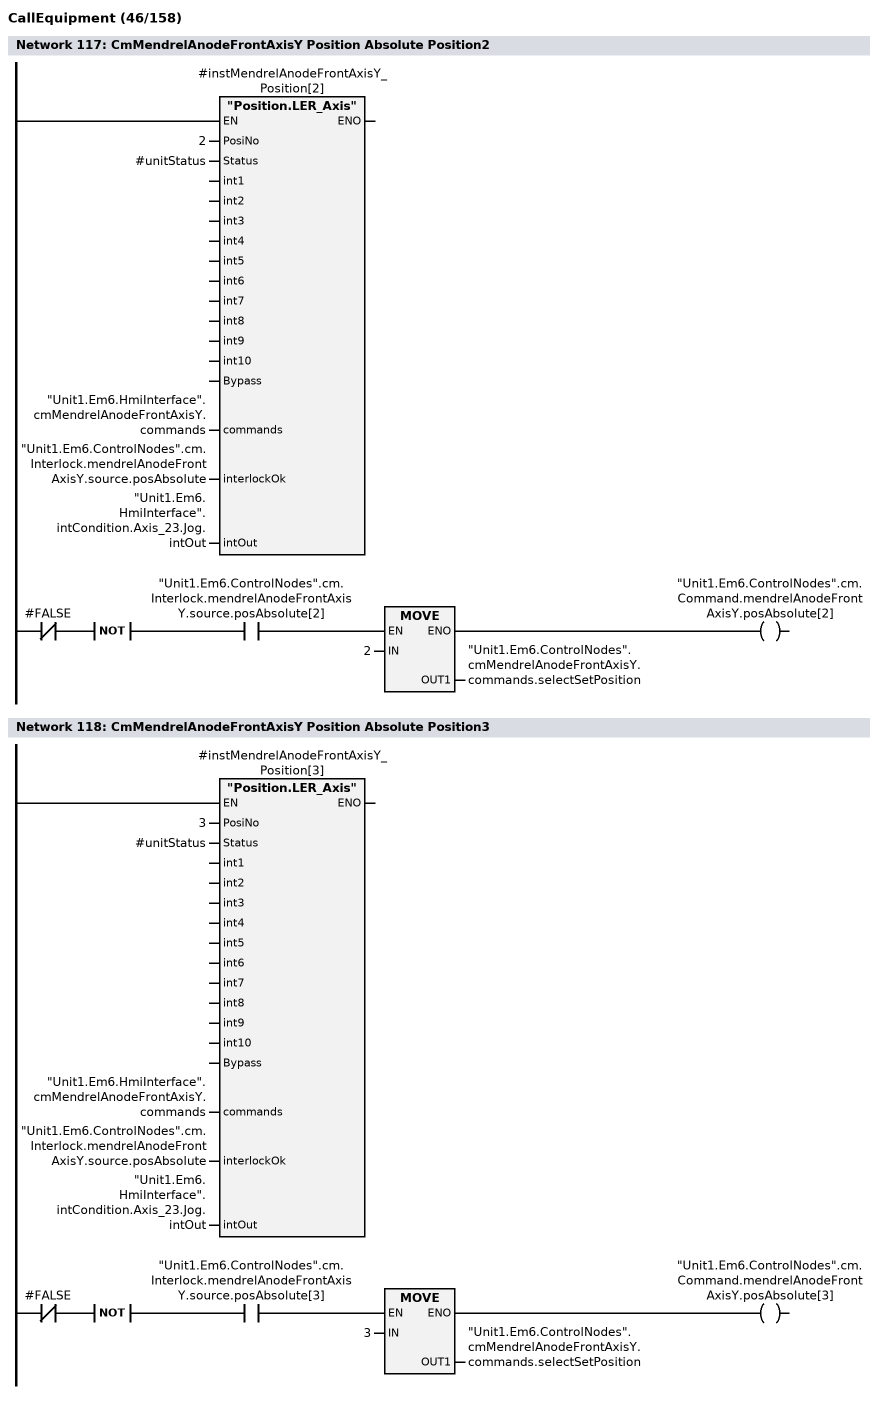
   RUNG wire#powerrail
      #instMendrelAnodeFrontAxisY_Position[2](PosiNo := 2, Status := #unitStatus, int1 :=, int2 :=, int3 :=, int4 :=, int5 :=, int6 :=, int7 :=, int8 :=, int9 :=, int10 :=, Bypass :=, commands := "Unit1.Em6.HmiInterface".cmMendrelAnodeFrontAxisY.commands, interlockOk := "Unit1.Em6.ControlNodes".cm.Interlock.mendrelAnodeFrontAxisY.source.posAbsolute, intOut := "Unit1.Em6.HmiInterface".intCondition.Axis_23.Jog.intOut)
   END_RUNG
   RUNG wire#powerrail
      I_Contact( #FALSE )
      Not()
      Contact( "Unit1.Em6.ControlNodes".cm.Interlock.mendrelAnodeFrontAxisY.source.posAbsolute[2] )
      Move(in := 2, out1 => "Unit1.Em6.ControlNodes".cmMendrelAnodeFrontAxisY.commands.selectSetPosition)
      Coil( "Unit1.Em6.ControlNodes".cm.Command.mendrelAnodeFrontAxisY.posAbsolute[2] )
   END_RUNG
   // the same network as SCL:
   #instMendrelAnodeFrontAxisY_Position[2](PosiNo := 2,   // "Position.LER_Axis"
                           Status := #unitStatus,
                           commands := "Unit1.Em6.HmiInterface".cmMendrelAnodeFrontAxisY.commands,
                           interlockOk := "Unit1.Em6.ControlNodes".cm.Interlock.mendrelAnodeFrontAxisY.source.posAbsolute,
                           intOut := "Unit1.Em6.HmiInterface".intCondition.Axis_23.Jog.intOut);
   #_w1 := NOT (NOT #FALSE) AND "Unit1.Em6.ControlNodes".cm.Interlock.mendrelAnodeFrontAxisY.source.posAbsolute[2];
   IF #_w1 THEN "Unit1.Em6.ControlNodes".cmMendrelAnodeFrontAxisY.commands.selectSetPosition := 2; END_IF;
   "Unit1.Em6.ControlNodes".cm.Command.mendrelAnodeFrontAxisY.posAbsolute[2] := #_w1;
END_REGION

REGION Network 118: CmMendrelAnodeFrontAxisY Position Absolute Position3
   RUNG wire#powerrail
      #instMendrelAnodeFrontAxisY_Position[3](PosiNo := 3, Status := #unitStatus, int1 :=, int2 :=, int3 :=, int4 :=, int5 :=, int6 :=, int7 :=, int8 :=, int9 :=, int10 :=, Bypass :=, commands := "Unit1.Em6.HmiInterface".cmMendrelAnodeFrontAxisY.commands, interlockOk := "Unit1.Em6.ControlNodes".cm.Interlock.mendrelAnodeFrontAxisY.source.posAbsolute, intOut := "Unit1.Em6.HmiInterface".intCondition.Axis_23.Jog.intOut)
   END_RUNG
   RUNG wire#powerrail
      I_Contact( #FALSE )
      Not()
      Contact( "Unit1.Em6.ControlNodes".cm.Interlock.mendrelAnodeFrontAxisY.source.posAbsolute[3] )
      Move(in := 3, out1 => "Unit1.Em6.ControlNodes".cmMendrelAnodeFrontAxisY.commands.selectSetPosition)
      Coil( "Unit1.Em6.ControlNodes".cm.Command.mendrelAnodeFrontAxisY.posAbsolute[3] )
   END_RUNG
   // the same network as SCL:
   #instMendrelAnodeFrontAxisY_Position[3](PosiNo := 3,   // "Position.LER_Axis"
                           Status := #unitStatus,
                           commands := "Unit1.Em6.HmiInterface".cmMendrelAnodeFrontAxisY.commands,
                           interlockOk := "Unit1.Em6.ControlNodes".cm.Interlock.mendrelAnodeFrontAxisY.source.posAbsolute,
                           intOut := "Unit1.Em6.HmiInterface".intCondition.Axis_23.Jog.intOut);
   #_w1 := NOT (NOT #FALSE) AND "Unit1.Em6.ControlNodes".cm.Interlock.mendrelAnodeFrontAxisY.source.posAbsolute[3];
   IF #_w1 THEN "Unit1.Em6.ControlNodes".cmMendrelAnodeFrontAxisY.commands.selectSetPosition := 3; END_IF;
   "Unit1.Em6.ControlNodes".cm.Command.mendrelAnodeFrontAxisY.posAbsolute[3] := #_w1;
END_REGION

REGION Network 119: CmMendrelAnodeFrontAxisY Position Absolute Position4
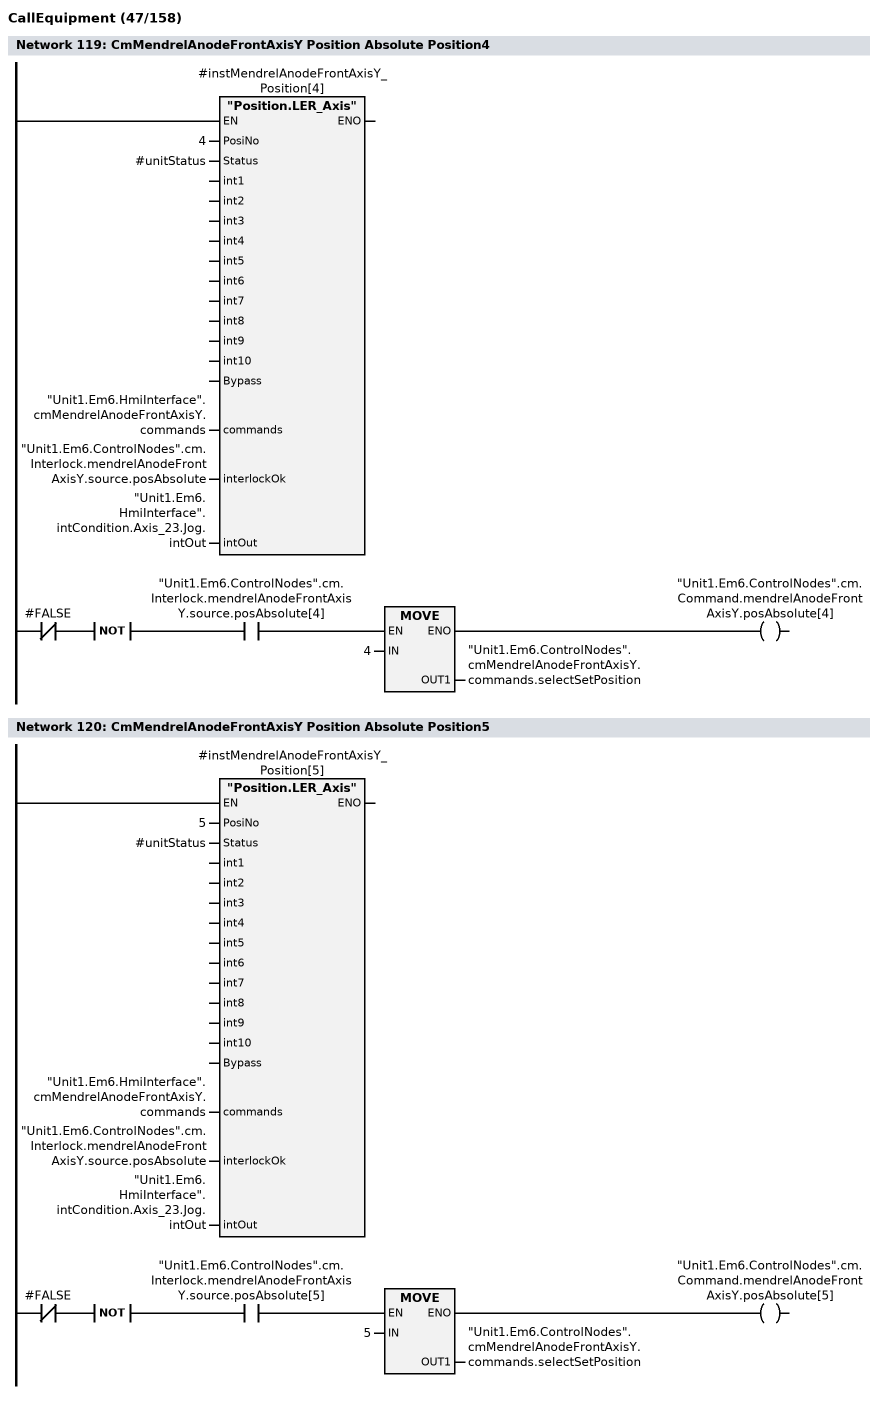
   RUNG wire#powerrail
      #instMendrelAnodeFrontAxisY_Position[4](PosiNo := 4, Status := #unitStatus, int1 :=, int2 :=, int3 :=, int4 :=, int5 :=, int6 :=, int7 :=, int8 :=, int9 :=, int10 :=, Bypass :=, commands := "Unit1.Em6.HmiInterface".cmMendrelAnodeFrontAxisY.commands, interlockOk := "Unit1.Em6.ControlNodes".cm.Interlock.mendrelAnodeFrontAxisY.source.posAbsolute, intOut := "Unit1.Em6.HmiInterface".intCondition.Axis_23.Jog.intOut)
   END_RUNG
   RUNG wire#powerrail
      I_Contact( #FALSE )
      Not()
      Contact( "Unit1.Em6.ControlNodes".cm.Interlock.mendrelAnodeFrontAxisY.source.posAbsolute[4] )
      Move(in := 4, out1 => "Unit1.Em6.ControlNodes".cmMendrelAnodeFrontAxisY.commands.selectSetPosition)
      Coil( "Unit1.Em6.ControlNodes".cm.Command.mendrelAnodeFrontAxisY.posAbsolute[4] )
   END_RUNG
   // the same network as SCL:
   #instMendrelAnodeFrontAxisY_Position[4](PosiNo := 4,   // "Position.LER_Axis"
                           Status := #unitStatus,
                           commands := "Unit1.Em6.HmiInterface".cmMendrelAnodeFrontAxisY.commands,
                           interlockOk := "Unit1.Em6.ControlNodes".cm.Interlock.mendrelAnodeFrontAxisY.source.posAbsolute,
                           intOut := "Unit1.Em6.HmiInterface".intCondition.Axis_23.Jog.intOut);
   #_w1 := NOT (NOT #FALSE) AND "Unit1.Em6.ControlNodes".cm.Interlock.mendrelAnodeFrontAxisY.source.posAbsolute[4];
   IF #_w1 THEN "Unit1.Em6.ControlNodes".cmMendrelAnodeFrontAxisY.commands.selectSetPosition := 4; END_IF;
   "Unit1.Em6.ControlNodes".cm.Command.mendrelAnodeFrontAxisY.posAbsolute[4] := #_w1;
END_REGION

REGION Network 120: CmMendrelAnodeFrontAxisY Position Absolute Position5
   RUNG wire#powerrail
      #instMendrelAnodeFrontAxisY_Position[5](PosiNo := 5, Status := #unitStatus, int1 :=, int2 :=, int3 :=, int4 :=, int5 :=, int6 :=, int7 :=, int8 :=, int9 :=, int10 :=, Bypass :=, commands := "Unit1.Em6.HmiInterface".cmMendrelAnodeFrontAxisY.commands, interlockOk := "Unit1.Em6.ControlNodes".cm.Interlock.mendrelAnodeFrontAxisY.source.posAbsolute, intOut := "Unit1.Em6.HmiInterface".intCondition.Axis_23.Jog.intOut)
   END_RUNG
   RUNG wire#powerrail
      I_Contact( #FALSE )
      Not()
      Contact( "Unit1.Em6.ControlNodes".cm.Interlock.mendrelAnodeFrontAxisY.source.posAbsolute[5] )
      Move(in := 5, out1 => "Unit1.Em6.ControlNodes".cmMendrelAnodeFrontAxisY.commands.selectSetPosition)
      Coil( "Unit1.Em6.ControlNodes".cm.Command.mendrelAnodeFrontAxisY.posAbsolute[5] )
   END_RUNG
   // the same network as SCL:
   #instMendrelAnodeFrontAxisY_Position[5](PosiNo := 5,   // "Position.LER_Axis"
                           Status := #unitStatus,
                           commands := "Unit1.Em6.HmiInterface".cmMendrelAnodeFrontAxisY.commands,
                           interlockOk := "Unit1.Em6.ControlNodes".cm.Interlock.mendrelAnodeFrontAxisY.source.posAbsolute,
                           intOut := "Unit1.Em6.HmiInterface".intCondition.Axis_23.Jog.intOut);
   #_w1 := NOT (NOT #FALSE) AND "Unit1.Em6.ControlNodes".cm.Interlock.mendrelAnodeFrontAxisY.source.posAbsolute[5];
   IF #_w1 THEN "Unit1.Em6.ControlNodes".cmMendrelAnodeFrontAxisY.commands.selectSetPosition := 5; END_IF;
   "Unit1.Em6.ControlNodes".cm.Command.mendrelAnodeFrontAxisY.posAbsolute[5] := #_w1;
END_REGION

REGION Network 121: CmMendrelAnodeFrontAxisY Summary Command
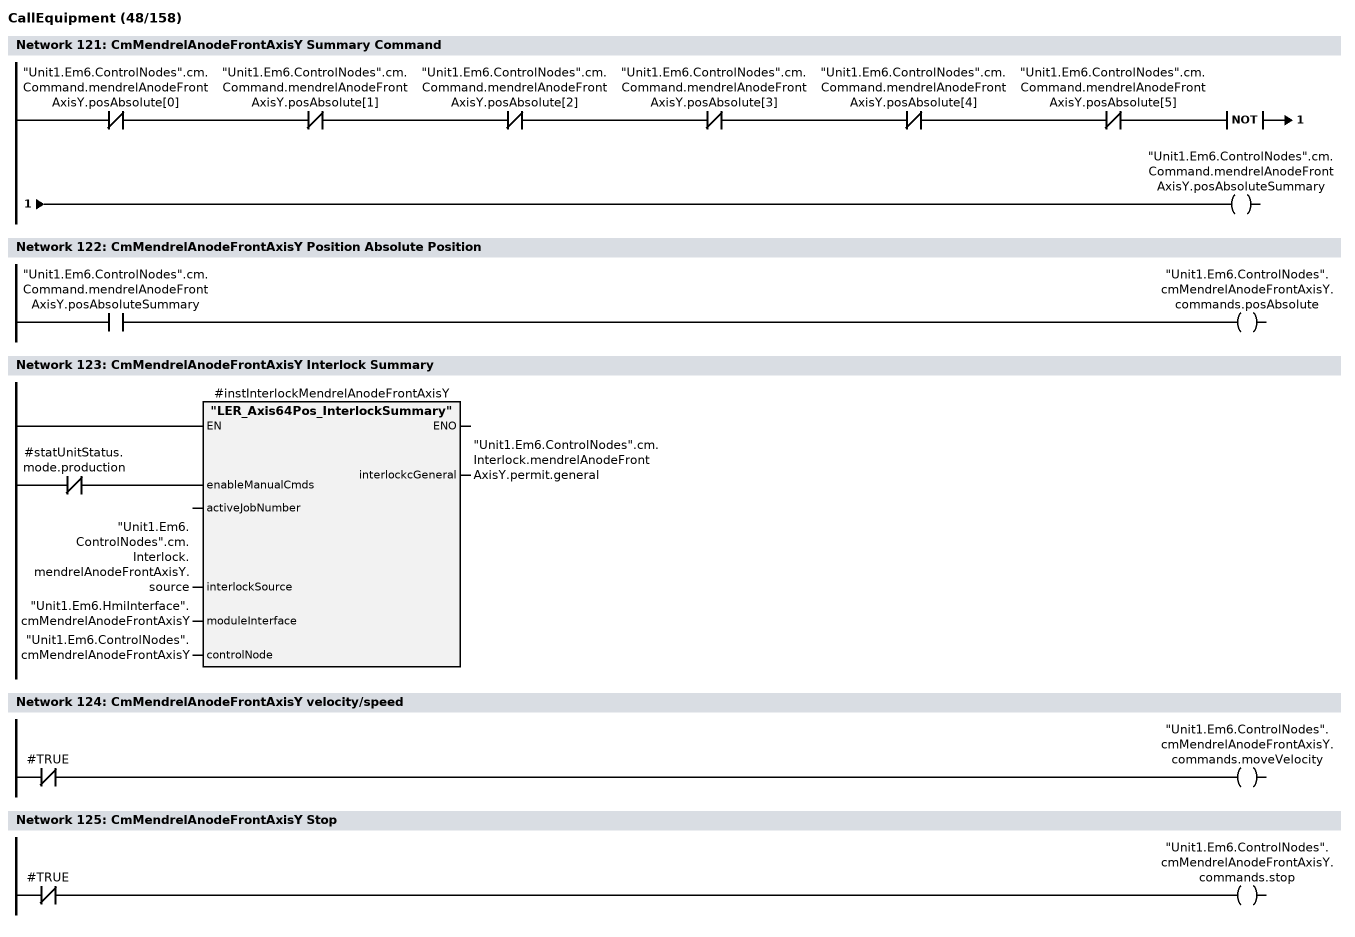
   RUNG wire#powerrail
      I_Contact( "Unit1.Em6.ControlNodes".cm.Command.mendrelAnodeFrontAxisY.posAbsolute[0] )
      I_Contact( "Unit1.Em6.ControlNodes".cm.Command.mendrelAnodeFrontAxisY.posAbsolute[1] )
      I_Contact( "Unit1.Em6.ControlNodes".cm.Command.mendrelAnodeFrontAxisY.posAbsolute[2] )
      I_Contact( "Unit1.Em6.ControlNodes".cm.Command.mendrelAnodeFrontAxisY.posAbsolute[3] )
      I_Contact( "Unit1.Em6.ControlNodes".cm.Command.mendrelAnodeFrontAxisY.posAbsolute[4] )
      I_Contact( "Unit1.Em6.ControlNodes".cm.Command.mendrelAnodeFrontAxisY.posAbsolute[5] )
      Not()
      Coil( "Unit1.Em6.ControlNodes".cm.Command.mendrelAnodeFrontAxisY.posAbsoluteSummary )
   END_RUNG
   // the same network as SCL:
   "Unit1.Em6.ControlNodes".cm.Command.mendrelAnodeFrontAxisY.posAbsoluteSummary := NOT (NOT "Unit1.Em6.ControlNodes".cm.Command.mendrelAnodeFrontAxisY.posAbsolute[0] AND NOT "Unit1.Em6.ControlNodes".cm.Command.mendrelAnodeFrontAxisY.posAbsolute[1] AND NOT "Unit1.Em6.ControlNodes".cm.Command.mendrelAnodeFrontAxisY.posAbsolute[2] AND NOT "Unit1.Em6.ControlNodes".cm.Command.mendrelAnodeFrontAxisY.posAbsolute[3] AND NOT "Unit1.Em6.ControlNodes".cm.Command.mendrelAnodeFrontAxisY.posAbsolute[4] AND NOT "Unit1.Em6.ControlNodes".cm.Command.mendrelAnodeFrontAxisY.posAbsolute[5]);
END_REGION

REGION Network 122: CmMendrelAnodeFrontAxisY Position Absolute Position
   RUNG wire#powerrail
      Contact( "Unit1.Em6.ControlNodes".cm.Command.mendrelAnodeFrontAxisY.posAbsoluteSummary )
      Coil( "Unit1.Em6.ControlNodes".cmMendrelAnodeFrontAxisY.commands.posAbsolute )
   END_RUNG
   // the same network as SCL:
   "Unit1.Em6.ControlNodes".cmMendrelAnodeFrontAxisY.commands.posAbsolute := "Unit1.Em6.ControlNodes".cm.Command.mendrelAnodeFrontAxisY.posAbsoluteSummary;
END_REGION

REGION Network 123: CmMendrelAnodeFrontAxisY Interlock Summary
   RUNG wire#powerrail
      #instInterlockMendrelAnodeFrontAxisY(enableManualCmds := wire#w1, activeJobNumber :=, interlockSource := "Unit1.Em6.ControlNodes".cm.Interlock.mendrelAnodeFrontAxisY.source, moduleInterface := "Unit1.Em6.HmiInterface".cmMendrelAnodeFrontAxisY, controlNode := "Unit1.Em6.ControlNodes".cmMendrelAnodeFrontAxisY, interlockcGeneral => "Unit1.Em6.ControlNodes".cm.Interlock.mendrelAnodeFrontAxisY.permit.general)
   END_RUNG
   RUNG wire#powerrail
      I_Contact( #statUnitStatus.mode.production )
   END_RUNG wire#w1
   // the same network as SCL:
   #instInterlockMendrelAnodeFrontAxisY(enableManualCmds := NOT #statUnitStatus.mode.production,   // "LER_Axis64Pos_InterlockSummary"
                           interlockSource := "Unit1.Em6.ControlNodes".cm.Interlock.mendrelAnodeFrontAxisY.source,
                           moduleInterface := "Unit1.Em6.HmiInterface".cmMendrelAnodeFrontAxisY,
                           controlNode := "Unit1.Em6.ControlNodes".cmMendrelAnodeFrontAxisY,
                           interlockcGeneral => "Unit1.Em6.ControlNodes".cm.Interlock.mendrelAnodeFrontAxisY.permit.general);
END_REGION

REGION Network 124: CmMendrelAnodeFrontAxisY velocity/speed
   RUNG wire#powerrail
      I_Contact( #TRUE )
      Coil( "Unit1.Em6.ControlNodes".cmMendrelAnodeFrontAxisY.commands.moveVelocity )
   END_RUNG
   // the same network as SCL:
   "Unit1.Em6.ControlNodes".cmMendrelAnodeFrontAxisY.commands.moveVelocity := NOT #TRUE;
END_REGION

REGION Network 125: CmMendrelAnodeFrontAxisY Stop
   RUNG wire#powerrail
      I_Contact( #TRUE )
      Coil( "Unit1.Em6.ControlNodes".cmMendrelAnodeFrontAxisY.commands.stop )
   END_RUNG
   // the same network as SCL:
   "Unit1.Em6.ControlNodes".cmMendrelAnodeFrontAxisY.commands.stop := NOT #TRUE;
END_REGION

REGION Network 126: Call CM Anode Mandrel Front Y-Axis (LBC_Axis64Pos)
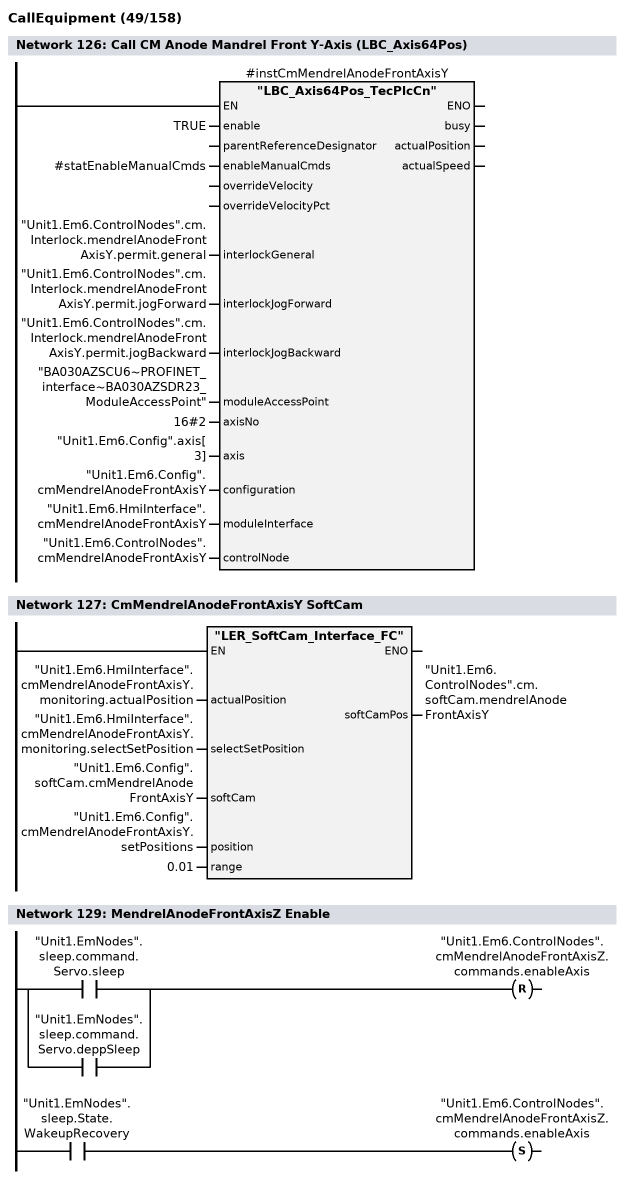
   RUNG wire#powerrail
      #instCmMendrelAnodeFrontAxisY(enable := TRUE, parentReferenceDesignator :=, enableManualCmds := #statEnableManualCmds, overrideVelocity :=, overrideVelocityPct :=, interlockGeneral := "Unit1.Em6.ControlNodes".cm.Interlock.mendrelAnodeFrontAxisY.permit.general, interlockJogForward := "Unit1.Em6.ControlNodes".cm.Interlock.mendrelAnodeFrontAxisY.permit.jogForward, interlockJogBackward := "Unit1.Em6.ControlNodes".cm.Interlock.mendrelAnodeFrontAxisY.permit.jogBackward, moduleAccessPoint := "BA030AZSCU6~PROFINET_interface~BA030AZSDR23_ModuleAccessPoint", axisNo := 16#2, axis := "Unit1.Em6.Config".axis[3], configuration := "Unit1.Em6.Config".cmMendrelAnodeFrontAxisY, moduleInterface := "Unit1.Em6.HmiInterface".cmMendrelAnodeFrontAxisY, controlNode := "Unit1.Em6.ControlNodes".cmMendrelAnodeFrontAxisY, busy =>, actualPosition =>, actualSpeed =>)
   END_RUNG
   // the same network as SCL:
   #instCmMendrelAnodeFrontAxisY(enable := TRUE,   // "LBC_Axis64Pos_TecPlcCn"
                           enableManualCmds := #statEnableManualCmds,
                           interlockGeneral := "Unit1.Em6.ControlNodes".cm.Interlock.mendrelAnodeFrontAxisY.permit.general,
                           interlockJogForward := "Unit1.Em6.ControlNodes".cm.Interlock.mendrelAnodeFrontAxisY.permit.jogForward,
                           interlockJogBackward := "Unit1.Em6.ControlNodes".cm.Interlock.mendrelAnodeFrontAxisY.permit.jogBackward,
                           moduleAccessPoint := "BA030AZSCU6~PROFINET_interface~BA030AZSDR23_ModuleAccessPoint",
                           axisNo := 16#2,
                           axis := "Unit1.Em6.Config".axis[3],
                           configuration := "Unit1.Em6.Config".cmMendrelAnodeFrontAxisY,
                           moduleInterface := "Unit1.Em6.HmiInterface".cmMendrelAnodeFrontAxisY,
                           controlNode := "Unit1.Em6.ControlNodes".cmMendrelAnodeFrontAxisY);
END_REGION

REGION Network 127: CmMendrelAnodeFrontAxisY SoftCam
   RUNG wire#powerrail
      "LER_SoftCam_Interface_FC"(actualPosition := "Unit1.Em6.HmiInterface".cmMendrelAnodeFrontAxisY.monitoring.actualPosition, selectSetPosition := "Unit1.Em6.HmiInterface".cmMendrelAnodeFrontAxisY.monitoring.selectSetPosition, softCam := "Unit1.Em6.Config".softCam.cmMendrelAnodeFrontAxisY, position := "Unit1.Em6.Config".cmMendrelAnodeFrontAxisY.setPositions, range := 0.01, softCamPos => "Unit1.Em6.ControlNodes".cm.softCam.mendrelAnodeFrontAxisY)
   END_RUNG
   // the same network as SCL:
   "LER_SoftCam_Interface_FC"(actualPosition := "Unit1.Em6.HmiInterface".cmMendrelAnodeFrontAxisY.monitoring.actualPosition,
                           selectSetPosition := "Unit1.Em6.HmiInterface".cmMendrelAnodeFrontAxisY.monitoring.selectSetPosition,
                           softCam := "Unit1.Em6.Config".softCam.cmMendrelAnodeFrontAxisY,
                           position := "Unit1.Em6.Config".cmMendrelAnodeFrontAxisY.setPositions,
                           range := 0.01,
                           softCamPos => "Unit1.Em6.ControlNodes".cm.softCam.mendrelAnodeFrontAxisY);
END_REGION

REGION Network 129: MendrelAnodeFrontAxisZ Enable
   RUNG wire#powerrail
      Contact( "Unit1.EmNodes".sleep.command.Servo.sleep )
      wire#w1
      R_Coil( "Unit1.Em6.ControlNodes".cmMendrelAnodeFrontAxisZ.commands.enableAxis )
   END_RUNG
   RUNG wire#powerrail
      Contact( "Unit1.EmNodes".sleep.command.Servo.deppSleep )
   END_RUNG wire#w1
   RUNG wire#powerrail
      Contact( "Unit1.EmNodes".sleep.State.WakeupRecovery )
      S_Coil( "Unit1.Em6.ControlNodes".cmMendrelAnodeFrontAxisZ.commands.enableAxis )
   END_RUNG
   // the same network as SCL:
   IF "Unit1.EmNodes".sleep.command.Servo.sleep OR "Unit1.EmNodes".sleep.command.Servo.deppSleep THEN
       "Unit1.Em6.ControlNodes".cmMendrelAnodeFrontAxisZ.commands.enableAxis := FALSE;
   END_IF;
   IF "Unit1.EmNodes".sleep.State.WakeupRecovery THEN
       "Unit1.Em6.ControlNodes".cmMendrelAnodeFrontAxisZ.commands.enableAxis := TRUE;
   END_IF;
END_REGION

REGION Network 130: CmMendrelAnodeFrontAxisZ Home
